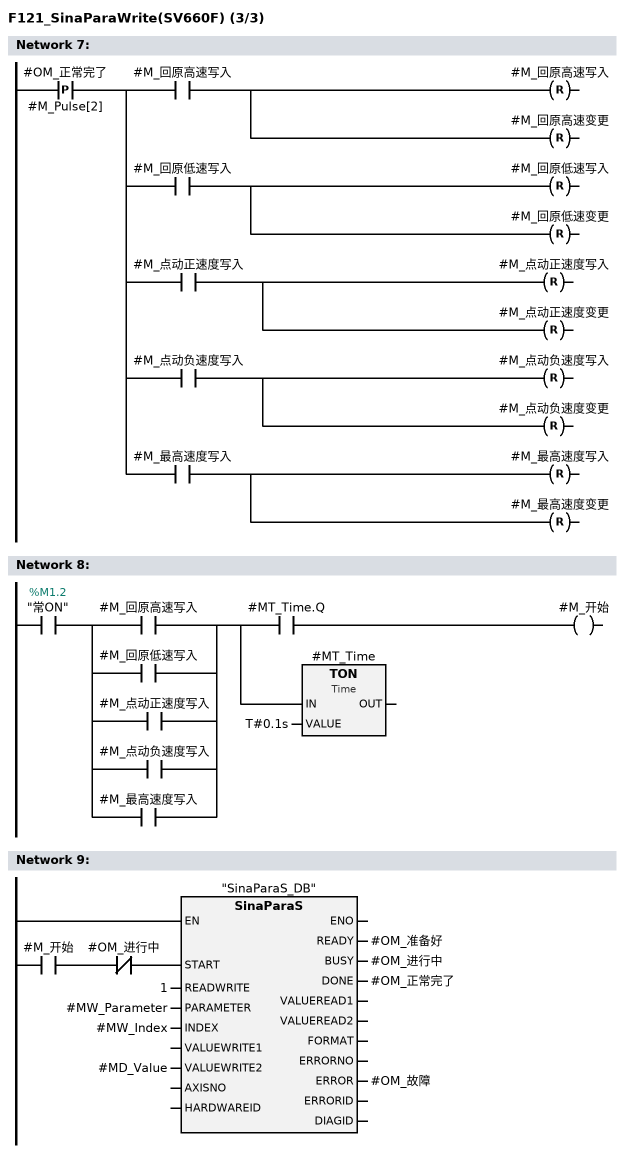
   RUNG wire#powerrail
      P_Contact(operand := #OM_正常完了, bit := #M_Pulse[2])
      wire#w1
      Contact( #M_回原高速写入 )
      wire#w2
      R_Coil( #M_回原高速写入 )
   END_RUNG
   RUNG wire#w2
      R_Coil( #M_回原高速变更 )
   END_RUNG
   RUNG wire#w1
      Contact( #M_回原低速写入 )
      wire#w3
      R_Coil( #M_回原低速写入 )
   END_RUNG
   RUNG wire#w3
      R_Coil( #M_回原低速变更 )
   END_RUNG
   RUNG wire#w1
      Contact( #M_点动正速度写入 )
      wire#w4
      R_Coil( #M_点动正速度写入 )
   END_RUNG
   RUNG wire#w4
      R_Coil( #M_点动正速度变更 )
   END_RUNG
   RUNG wire#w1
      Contact( #M_点动负速度写入 )
      wire#w5
      R_Coil( #M_点动负速度写入 )
   END_RUNG
   RUNG wire#w5
      R_Coil( #M_点动负速度变更 )
   END_RUNG
   RUNG wire#w1
      Contact( #M_最高速度写入 )
      wire#w6
      R_Coil( #M_最高速度写入 )
   END_RUNG
   RUNG wire#w6
      R_Coil( #M_最高速度变更 )
   END_RUNG
   // the same network as SCL:
   #_w1 := #OM_正常完了 AND NOT #M_Pulse[2];   // rising edge of #OM_正常完了
   #M_Pulse[2] := #OM_正常完了;
   #_w2 := #_w1 AND #M_回原高速写入;
   IF #_w2 THEN
       #M_回原高速写入 := FALSE;
       #M_回原高速变更 := FALSE;
   END_IF;
   #_w3 := #_w1 AND #M_回原低速写入;
   IF #_w3 THEN
       #M_回原低速写入 := FALSE;
       #M_回原低速变更 := FALSE;
   END_IF;
   #_w4 := #_w1 AND #M_点动正速度写入;
   IF #_w4 THEN
       #M_点动正速度写入 := FALSE;
       #M_点动正速度变更 := FALSE;
   END_IF;
   #_w5 := #_w1 AND #M_点动负速度写入;
   IF #_w5 THEN
       #M_点动负速度写入 := FALSE;
       #M_点动负速度变更 := FALSE;
   END_IF;
   #_w6 := #_w1 AND #M_最高速度写入;
   IF #_w6 THEN
       #M_最高速度写入 := FALSE;
       #M_最高速度变更 := FALSE;
   END_IF;
END_REGION

REGION Network 8
   #_w1 := "常ON" AND (#M_回原高速写入 OR #M_回原低速写入 OR #M_点动正速度写入 OR #M_点动负速度写入 OR #M_最高速度写入);
   #M_开始 := #_w1 AND #MT_Time.Q;
   #MT_Time.TON(IN := #_w1, PT := T#0.1s);   // TON coil
END_REGION

REGION Network 9
   RUNG wire#powerrail
      "SinaParaS_DB".SinaParaS(Start := wire#w1, ReadWrite := 1, Parameter := #MW_Parameter, Index := #MW_Index, ValueWrite1 :=, ValueWrite2 := #MD_Value, AxisNo :=, hardwareId :=, Ready => #OM_准备好, Busy => #OM_进行中, Done => #OM_正常完了, ValueRead1 =>, ValueRead2 =>, Format =>, ErrorNo =>, Error => #OM_故障, ErrorId =>, DiagId =>)
   END_RUNG
   RUNG wire#powerrail
      Contact( #M_开始 )
      I_Contact( #OM_进行中 )
   END_RUNG wire#w1
   // the same network as SCL:
   "SinaParaS_DB"(Start := #M_开始 AND NOT #OM_进行中,   // SinaParaS
                  ReadWrite := 1,
                  Parameter := #MW_Parameter,
                  Index := #MW_Index,
                  ValueWrite2 := #MD_Value,
                  Ready => #OM_准备好,
                  Busy => #OM_进行中,
                  Done => #OM_正常完了,
                  Error => #OM_故障);
END_REGION
END_FUNCTION_BLOCK

FUNCTION_BLOCK "F120_SinaPos(SV660F)"   // FB120, LAD
{ S7_Optimized_Access := 'TRUE' }
VERSION : 0.1
// 2024/2/4:第一版本V1.0，作者:wang
// stored: AutoNumber false, IsIECCheckEnabled false, IsRetainMemResEnabled false, MemoryReserve 100, SetENOAutomatically false, UDAEnableTagReadback false
   VAR_INPUT
      IW_手动模式 { ExternalAccessible := 'False'; ExternalVisible := 'False'; ExternalWritable := 'False'} : Bool;
      IW_运行条件 { ExternalAccessible := 'False'; ExternalVisible := 'False'; ExternalWritable := 'False'} : Array[1..8] of Bool;
      IM_使能 { ExternalAccessible := 'False'; ExternalVisible := 'False'; ExternalWritable := 'False'} : Bool;
      IM_回零 { ExternalAccessible := 'False'; ExternalVisible := 'False'; ExternalWritable := 'False'} : Bool;
      IM_绝对定位 { ExternalAccessible := 'False'; ExternalVisible := 'False'; ExternalWritable := 'False'} : Bool;
      IM_相对定位 { ExternalAccessible := 'False'; ExternalVisible := 'False'; ExternalWritable := 'False'} : Bool;
      "IM_JOG+" { ExternalAccessible := 'False'; ExternalVisible := 'False'; ExternalWritable := 'False'} : Bool;
      "IM_JOG-" { ExternalAccessible := 'False'; ExternalVisible := 'False'; ExternalWritable := 'False'} : Bool;
      IM_故障复位 { ExternalAccessible := 'False'; ExternalVisible := 'False'; ExternalWritable := 'False'} : Bool;
      ID_目标位置 { ExternalAccessible := 'False'; ExternalVisible := 'False'; ExternalWritable := 'False'} : DInt;
      ID_目标速度 { ExternalAccessible := 'False'; ExternalVisible := 'False'; ExternalWritable := 'False'} : DInt;
      "IW_速度加减倍率%" { ExternalAccessible := 'False'; ExternalVisible := 'False'; ExternalWritable := 'False'} : Array[1..3] of Int;
      ID_ConfigEpos { ExternalAccessible := 'False'; ExternalVisible := 'False'; ExternalWritable := 'False'} : DWord;
      ID_111报文标识符 { ExternalAccessible := 'False'; ExternalVisible := 'False'; ExternalWritable := 'False'} : HW_IO;
   END_VAR
   VAR_OUTPUT
      OM_准备好了 : Bool;
      OM_动作中 : Bool;
      OM_回零完了 : Bool;
      OM_轴报警 : Bool;
      OM_轴错误 : Bool;
      OD_当前位置 : DInt;
      OD_当前速度 : DInt;
      OW_运行模式 : Int;
      OW_EPSW1 : Word;
      OW_EPSW2 : Word;
      OW_轴报警码 : Word;
      OW_轴错误码 : Word;
      OW_库错误码 : Int;
      OW_调用错误码 : Word;
   END_VAR
   VAR
      MT_StartChk : IEC_TIMER;   // 启动延迟
   END_VAR
   VAR_TEMP
      M_停止 : Bool;
      M_暂停 : Bool;
      M_JOG指令 : Bool;
      M_回零指令 : Bool;
      M_绝对定位指令 : Bool;
      M_相对定位指令 : Bool;
      M_回零定位完Pls : Bool;
      M_绝对定位完Pls : Bool;
      M_相对定位完Pls : Bool;
      M_启动 : Bool;
      M_定位完了 : Bool;
      W_运行模式 : Int;
      M_Pulse : Array[1..20] of Bool;
      M_SerState : Bool;   // 伺服正常
      M_Busy : Bool;   // 伺服忙
      M_FLS_SW : Bool;   // 正极限
      M_RLS_SW : Bool;   // 负极限
   END_VAR
   // // IW_运行条件[1] : 共同条件
   // // IW_运行条件[2] : 回零条件
   // // IW_运行条件[3] : JOG正条件
   // // IW_运行条件[4] : JOG负条件
   // // IW_运行条件[5] : 定位正条件
   // // IW_运行条件[6] : 定位负条件
   // // IW_运行条件[7] : 预留
   // // IW_运行条件[8] : 预留
   VAR_TEMP   // added for the SCL form of the ladder/FBD networks
      _w1 : Bool;
      _w2 : Bool;
      _w3 : Bool;
      _w4 : Bool;
   END_VAR
BEGIN

REGION Network 1: 伺服状态条件
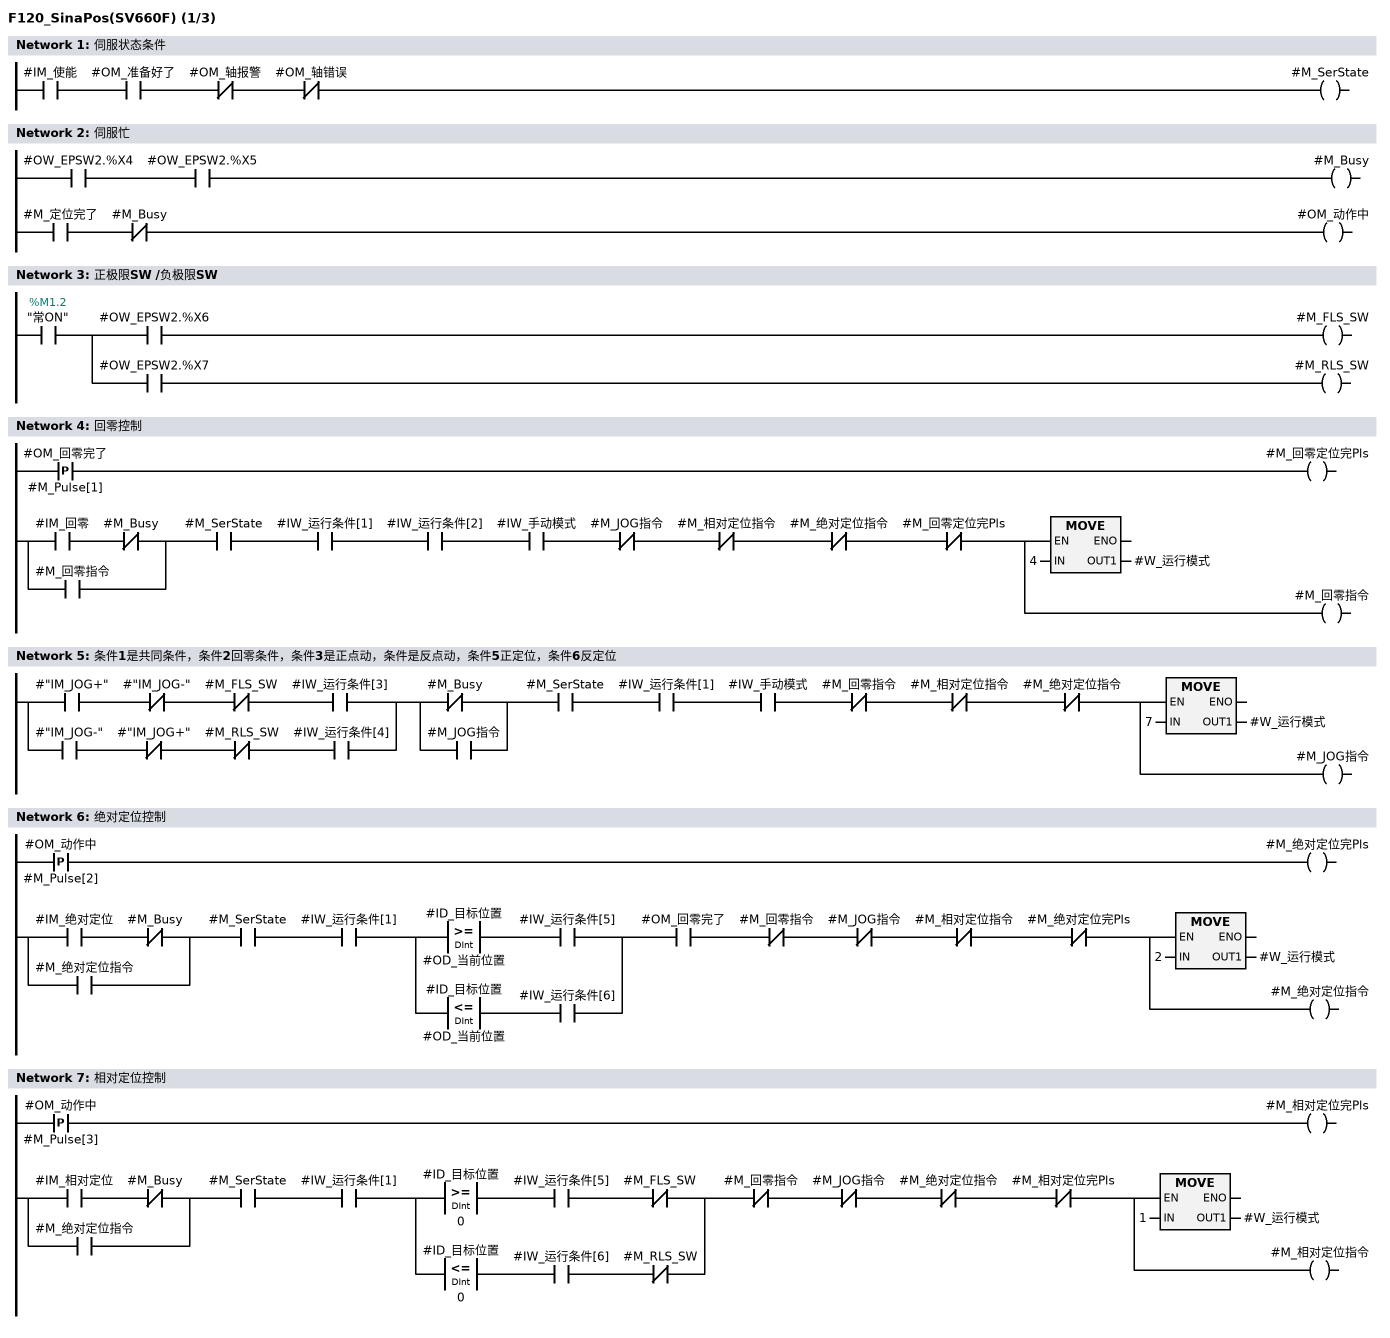
   RUNG wire#powerrail
      Contact( #IM_使能 )
      Contact( #OM_准备好了 )
      I_Contact( #OM_轴报警 )
      I_Contact( #OM_轴错误 )
      Coil( #M_SerState )
   END_RUNG
   // the same network as SCL:
   #M_SerState := #IM_使能 AND #OM_准备好了 AND NOT #OM_轴报警 AND NOT #OM_轴错误;
END_REGION

REGION Network 2: 伺服忙
   RUNG wire#powerrail
      Contact( #OW_EPSW2.%X4 )
      Contact( #OW_EPSW2.%X5 )
      Coil( #M_Busy )
   END_RUNG
   RUNG wire#powerrail
      Contact( #M_定位完了 )
      I_Contact( #M_Busy )
      Coil( #OM_动作中 )
   END_RUNG
   // the same network as SCL:
   #M_Busy := #OW_EPSW2.%X4 AND #OW_EPSW2.%X5;
   #OM_动作中 := #M_定位完了 AND NOT #M_Busy;
END_REGION

REGION Network 3: 正极限SW /负极限SW
   RUNG wire#powerrail
      Contact( "常ON" )
      wire#w1
      Contact( #OW_EPSW2.%X6 )
      Coil( #M_FLS_SW )
   END_RUNG
   RUNG wire#w1
      Contact( #OW_EPSW2.%X7 )
      Coil( #M_RLS_SW )
   END_RUNG
   // the same network as SCL:
   #M_FLS_SW := "常ON" AND #OW_EPSW2.%X6;
   #M_RLS_SW := "常ON" AND #OW_EPSW2.%X7;
END_REGION

REGION Network 4: 回零控制
   RUNG wire#powerrail
      P_Contact(operand := #OM_回零完了, bit := #M_Pulse[1])
      Coil( #M_回零定位完Pls )
   END_RUNG
   RUNG wire#powerrail
      Contact( #IM_回零 )
      I_Contact( #M_Busy )
      wire#w1
      Contact( #M_SerState )
      Contact( #IW_运行条件[1] )
      Contact( #IW_运行条件[2] )
      Contact( #IW_手动模式 )
      I_Contact( #M_JOG指令 )
      I_Contact( #M_相对定位指令 )
      I_Contact( #M_绝对定位指令 )
      I_Contact( #M_回零定位完Pls )
      wire#w2
      Move(in := 4, out1 => #W_运行模式)
   END_RUNG
   RUNG wire#powerrail
      Contact( #M_回零指令 )
   END_RUNG wire#w1
   RUNG wire#w2
      Coil( #M_回零指令 )
   END_RUNG
   // the same network as SCL:
   #_w1 := #OM_回零完了 AND NOT #M_Pulse[1];   // rising edge of #OM_回零完了
   #M_Pulse[1] := #OM_回零完了;
   #M_回零定位完Pls := #_w1;
   #_w2 := ((#IM_回零 AND NOT #M_Busy) OR #M_回零指令) AND #M_SerState AND #IW_运行条件[1] AND #IW_运行条件[2] AND #IW_手动模式 AND NOT #M_JOG指令 AND NOT #M_相对定位指令 AND NOT #M_绝对定位指令 AND NOT #M_回零定位完Pls;
   IF #_w2 THEN #W_运行模式 := 4; END_IF;
   #M_回零指令 := #_w2;
END_REGION

REGION Network 5: 条件1是共同条件，条件2回零条件，条件3是正点动，条件是反点动，条件5正定位，条件6反定位
   RUNG wire#powerrail
      Contact( #"IM_JOG+" )
      I_Contact( #"IM_JOG-" )
      I_Contact( #M_FLS_SW )
      Contact( #IW_运行条件[3] )
      wire#w1
      I_Contact( #M_Busy )
      wire#w2
      Contact( #M_SerState )
      Contact( #IW_运行条件[1] )
      Contact( #IW_手动模式 )
      I_Contact( #M_回零指令 )
      I_Contact( #M_相对定位指令 )
      I_Contact( #M_绝对定位指令 )
      wire#w3
      Move(in := 7, out1 => #W_运行模式)
   END_RUNG
   RUNG wire#powerrail
      Contact( #"IM_JOG-" )
      I_Contact( #"IM_JOG+" )
      I_Contact( #M_RLS_SW )
      Contact( #IW_运行条件[4] )
   END_RUNG wire#w1
   RUNG wire#w1
      Contact( #M_JOG指令 )
   END_RUNG wire#w2
   RUNG wire#w3
      Coil( #M_JOG指令 )
   END_RUNG
   // the same network as SCL:
   #_w1 := ((#"IM_JOG+" AND NOT #"IM_JOG-" AND NOT #M_FLS_SW AND #IW_运行条件[3]) OR (#"IM_JOG-" AND NOT #"IM_JOG+" AND NOT #M_RLS_SW AND #IW_运行条件[4])) AND (NOT #M_Busy OR #M_JOG指令) AND #M_SerState AND #IW_运行条件[1] AND #IW_手动模式 AND NOT #M_回零指令 AND NOT #M_相对定位指令 AND NOT #M_绝对定位指令;
   IF #_w1 THEN #W_运行模式 := 7; END_IF;
   #M_JOG指令 := #_w1;
END_REGION

REGION Network 6: 绝对定位控制
   RUNG wire#powerrail
      P_Contact(operand := #OM_动作中, bit := #M_Pulse[2])
      Coil( #M_绝对定位完Pls )
   END_RUNG
   RUNG wire#powerrail
      Contact( #IM_绝对定位 )
      I_Contact( #M_Busy )
      wire#w1
      Contact( #M_SerState )
      Contact( #IW_运行条件[1] )
      wire#w2
      { S7_Templates := "SrcType := DInt" } GE_Contact(in1 := #ID_目标位置, in2 := #OD_当前位置)
      Contact( #IW_运行条件[5] )
      wire#w3
      Contact( #OM_回零完了 )
      I_Contact( #M_回零指令 )
      I_Contact( #M_JOG指令 )
      I_Contact( #M_相对定位指令 )
      I_Contact( #M_绝对定位完Pls )
      wire#w4
      Move(in := 2, out1 => #W_运行模式)
   END_RUNG
   RUNG wire#powerrail
      Contact( #M_绝对定位指令 )
   END_RUNG wire#w1
   RUNG wire#w2
      { S7_Templates := "SrcType := DInt" } LE_Contact(in1 := #ID_目标位置, in2 := #OD_当前位置)
      Contact( #IW_运行条件[6] )
   END_RUNG wire#w3
   RUNG wire#w4
      Coil( #M_绝对定位指令 )
   END_RUNG
   // the same network as SCL:
   #_w1 := #OM_动作中 AND NOT #M_Pulse[2];   // rising edge of #OM_动作中
   #M_Pulse[2] := #OM_动作中;
   #M_绝对定位完Pls := #_w1;
   #_w2 := ((#IM_绝对定位 AND NOT #M_Busy) OR #M_绝对定位指令) AND #M_SerState AND #IW_运行条件[1] AND (((#ID_目标位置 >= #OD_当前位置) AND #IW_运行条件[5]) OR ((#ID_目标位置 <= #OD_当前位置) AND #IW_运行条件[6])) AND #OM_回零完了 AND NOT #M_回零指令 AND NOT #M_JOG指令 AND NOT #M_相对定位指令 AND NOT #M_绝对定位完Pls;
   IF #_w2 THEN #W_运行模式 := 2; END_IF;
   #M_绝对定位指令 := #_w2;
END_REGION

REGION Network 7: 相对定位控制
   RUNG wire#powerrail
      P_Contact(operand := #OM_动作中, bit := #M_Pulse[3])
      Coil( #M_相对定位完Pls )
   END_RUNG
   RUNG wire#powerrail
      Contact( #IM_相对定位 )
      I_Contact( #M_Busy )
      wire#w1
      Contact( #M_SerState )
      Contact( #IW_运行条件[1] )
      wire#w2
      { S7_Templates := "SrcType := DInt" } GE_Contact(in1 := #ID_目标位置, in2 := 0)
      Contact( #IW_运行条件[5] )
      I_Contact( #M_FLS_SW )
      wire#w3
      I_Contact( #M_回零指令 )
      I_Contact( #M_JOG指令 )
      I_Contact( #M_绝对定位指令 )
      I_Contact( #M_相对定位完Pls )
      wire#w4
      Move(in := 1, out1 => #W_运行模式)
   END_RUNG
   RUNG wire#powerrail
      Contact( #M_绝对定位指令 )
   END_RUNG wire#w1
   RUNG wire#w2
      { S7_Templates := "SrcType := DInt" } LE_Contact(in1 := #ID_目标位置, in2 := 0)
      Contact( #IW_运行条件[6] )
      I_Contact( #M_RLS_SW )
   END_RUNG wire#w3
   RUNG wire#w4
      Coil( #M_相对定位指令 )
   END_RUNG
   // the same network as SCL:
   #_w1 := #OM_动作中 AND NOT #M_Pulse[3];   // rising edge of #OM_动作中
   #M_Pulse[3] := #OM_动作中;
   #M_相对定位完Pls := #_w1;
   #_w2 := ((#IM_相对定位 AND NOT #M_Busy) OR #M_绝对定位指令) AND #M_SerState AND #IW_运行条件[1] AND (((#ID_目标位置 >= 0) AND #IW_运行条件[5] AND NOT #M_FLS_SW) OR ((#ID_目标位置 <= 0) AND #IW_运行条件[6] AND NOT #M_RLS_SW)) AND NOT #M_回零指令 AND NOT #M_JOG指令 AND NOT #M_绝对定位指令 AND NOT #M_相对定位完Pls;
   IF #_w2 THEN #W_运行模式 := 1; END_IF;
   #M_相对定位指令 := #_w2;
END_REGION

REGION Network 8: 控制启动
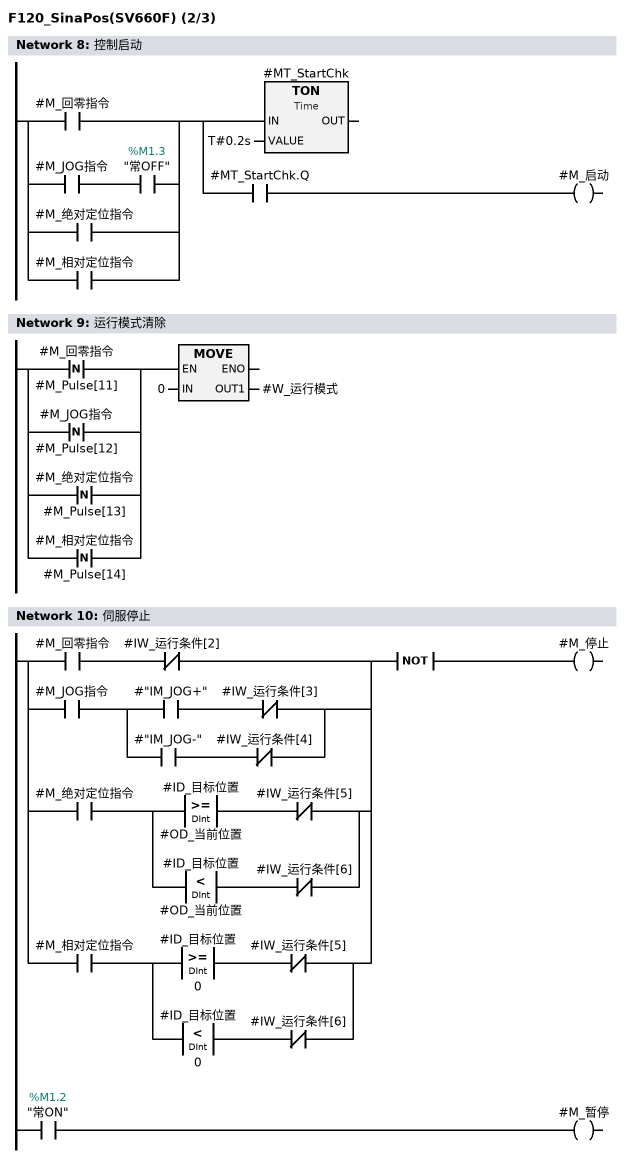
   #_w1 := #M_回零指令 OR (#M_JOG指令 AND "常OFF") OR #M_绝对定位指令 OR #M_相对定位指令;
   #MT_StartChk.TON(IN := #_w1, PT := T#0.2s);   // TON coil
   #M_启动 := #_w1 AND #MT_StartChk.Q;
END_REGION

REGION Network 9: 运行模式清除
   RUNG wire#powerrail
      N_Contact(operand := #M_回零指令, bit := #M_Pulse[11])
      wire#w1
      Move(in := 0, out1 => #W_运行模式)
   END_RUNG
   RUNG wire#powerrail
      N_Contact(operand := #M_JOG指令, bit := #M_Pulse[12])
   END_RUNG wire#w1
   RUNG wire#powerrail
      N_Contact(operand := #M_绝对定位指令, bit := #M_Pulse[13])
   END_RUNG wire#w1
   RUNG wire#powerrail
      N_Contact(operand := #M_相对定位指令, bit := #M_Pulse[14])
   END_RUNG wire#w1
   // the same network as SCL:
   #_w1 := NOT #M_回零指令 AND #M_Pulse[11];   // falling edge of #M_回零指令
   #M_Pulse[11] := #M_回零指令;
   #_w2 := NOT #M_JOG指令 AND #M_Pulse[12];   // falling edge of #M_JOG指令
   #M_Pulse[12] := #M_JOG指令;
   #_w3 := NOT #M_绝对定位指令 AND #M_Pulse[13];   // falling edge of #M_绝对定位指令
   #M_Pulse[13] := #M_绝对定位指令;
   #_w4 := NOT #M_相对定位指令 AND #M_Pulse[14];   // falling edge of #M_相对定位指令
   #M_Pulse[14] := #M_相对定位指令;
   IF #_w1 OR #_w2 OR #_w3 OR #_w4 THEN #W_运行模式 := 0; END_IF;
END_REGION

REGION Network 10: 伺服停止
   RUNG wire#powerrail
      Contact( #M_回零指令 )
      I_Contact( #IW_运行条件[2] )
      wire#w1
      Not()
      Coil( #M_停止 )
   END_RUNG
   RUNG wire#powerrail
      Contact( #M_JOG指令 )
      wire#w2
      Contact( #"IM_JOG+" )
      I_Contact( #IW_运行条件[3] )
   END_RUNG wire#w1
   RUNG wire#w2
      Contact( #"IM_JOG-" )
      I_Contact( #IW_运行条件[4] )
   END_RUNG wire#w1
   RUNG wire#powerrail
      Contact( #M_绝对定位指令 )
      wire#w3
      { S7_Templates := "SrcType := DInt" } GE_Contact(in1 := #ID_目标位置, in2 := #OD_当前位置)
      I_Contact( #IW_运行条件[5] )
   END_RUNG wire#w1
   RUNG wire#w3
      { S7_Templates := "SrcType := DInt" } LT_Contact(in1 := #ID_目标位置, in2 := #OD_当前位置)
      I_Contact( #IW_运行条件[6] )
   END_RUNG wire#w1
   RUNG wire#powerrail
      Contact( #M_相对定位指令 )
      wire#w4
      { S7_Templates := "SrcType := DInt" } GE_Contact(in1 := #ID_目标位置, in2 := 0)
      I_Contact( #IW_运行条件[5] )
   END_RUNG wire#w1
   RUNG wire#w4
      { S7_Templates := "SrcType := DInt" } LT_Contact(in1 := #ID_目标位置, in2 := 0)
      I_Contact( #IW_运行条件[6] )
   END_RUNG wire#w1
   RUNG wire#powerrail
      Contact( "常ON" )
      Coil( #M_暂停 )
   END_RUNG
   // the same network as SCL:
   #M_停止 := NOT ((#M_回零指令 AND NOT #IW_运行条件[2]) OR (#M_JOG指令 AND ((#"IM_JOG+" AND NOT #IW_运行条件[3]) OR (#"IM_JOG-" AND NOT #IW_运行条件[4]))) OR (#M_绝对定位指令 AND (((#ID_目标位置 >= #OD_当前位置) AND NOT #IW_运行条件[5]) OR ((#ID_目标位置 < #OD_当前位置) AND NOT #IW_运行条件[6]))) OR (#M_相对定位指令 AND (((#ID_目标位置 >= 0) AND NOT #IW_运行条件[5]) OR ((#ID_目标位置 < 0) AND NOT #IW_运行条件[6]))));
   #M_暂停 := "常ON";
END_REGION

REGION Network 11
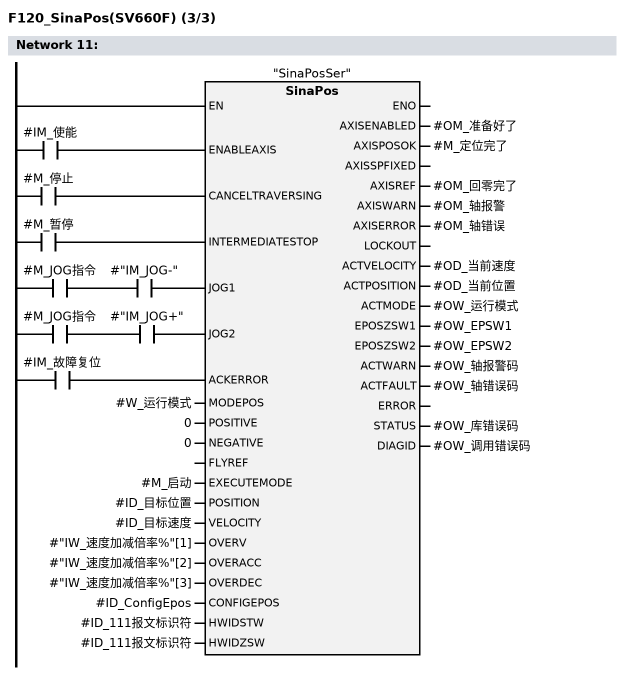
   RUNG wire#powerrail
      "SinaPosSer".SinaPos(EnableAxis := wire#w1, CancelTraversing := wire#w2, IntermediateStop := wire#w3, Jog1 := wire#w4, Jog2 := wire#w5, AckError := wire#w6, ModePos := #W_运行模式, Positive := 0, Negative := 0, FlyRef :=, ExecuteMode := #M_启动, Position := #ID_目标位置, Velocity := #ID_目标速度, OverV := #"IW_速度加减倍率%"[1], OverAcc := #"IW_速度加减倍率%"[2], OverDec := #"IW_速度加减倍率%"[3], ConfigEPos := #ID_ConfigEpos, HWIDSTW := #ID_111报文标识符, HWIDZSW := #ID_111报文标识符, AxisEnabled => #OM_准备好了, AxisPosOk => #M_定位完了, AxisSpFixed =>, AxisRef => #OM_回零完了, AxisWarn => #OM_轴报警, AxisError => #OM_轴错误, Lockout =>, ActVelocity => #OD_当前速度, ActPosition => #OD_当前位置, ActMode => #OW_运行模式, EPosZSW1 => #OW_EPSW1, EPosZSW2 => #OW_EPSW2, ActWarn => #OW_轴报警码, ActFault => #OW_轴错误码, Error =>, Status => #OW_库错误码, DiagId => #OW_调用错误码)
   END_RUNG
   RUNG wire#powerrail
      Contact( #IM_使能 )
   END_RUNG wire#w1
   RUNG wire#powerrail
      Contact( #M_停止 )
   END_RUNG wire#w2
   RUNG wire#powerrail
      Contact( #M_暂停 )
   END_RUNG wire#w3
   RUNG wire#powerrail
      Contact( #M_JOG指令 )
      Contact( #"IM_JOG-" )
   END_RUNG wire#w4
   RUNG wire#powerrail
      Contact( #M_JOG指令 )
      Contact( #"IM_JOG+" )
   END_RUNG wire#w5
   RUNG wire#powerrail
      Contact( #IM_故障复位 )
   END_RUNG wire#w6
   // the same network as SCL:
   "SinaPosSer"(EnableAxis := #IM_使能,   // SinaPos
                CancelTraversing := #M_停止,
                IntermediateStop := #M_暂停,
                Jog1 := #M_JOG指令 AND #"IM_JOG-",
                Jog2 := #M_JOG指令 AND #"IM_JOG+",
                AckError := #IM_故障复位,
                ModePos := #W_运行模式,
                Positive := 0,
                Negative := 0,
                ExecuteMode := #M_启动,
                Position := #ID_目标位置,
                Velocity := #ID_目标速度,
                OverV := #"IW_速度加减倍率%"[1],
                OverAcc := #"IW_速度加减倍率%"[2],
                OverDec := #"IW_速度加减倍率%"[3],
                ConfigEPos := #ID_ConfigEpos,
                HWIDSTW := #ID_111报文标识符,
                HWIDZSW := #ID_111报文标识符,
                AxisEnabled => #OM_准备好了,
                AxisPosOk => #M_定位完了,
                AxisRef => #OM_回零完了,
                AxisWarn => #OM_轴报警,
                AxisError => #OM_轴错误,
                ActVelocity => #OD_当前速度,
                ActPosition => #OD_当前位置,
                ActMode => #OW_运行模式,
                EPosZSW1 => #OW_EPSW1,
                EPosZSW2 => #OW_EPSW2,
                ActWarn => #OW_轴报警码,
                ActFault => #OW_轴错误码,
                Status => #OW_库错误码,
                DiagId => #OW_调用错误码);
END_REGION
END_FUNCTION_BLOCK

FUNCTION_BLOCK "K08_指示灯"   // FB8, LAD
{ S7_Optimized_Access := 'TRUE' }
VERSION : 0.1
// stored: AutoNumber false, IsIECCheckEnabled false, IsRetainMemResEnabled false, MemoryReserve 100, SetENOAutomatically false, UDAEnableTagReadback false
BEGIN

REGION Network 1: 自动灯
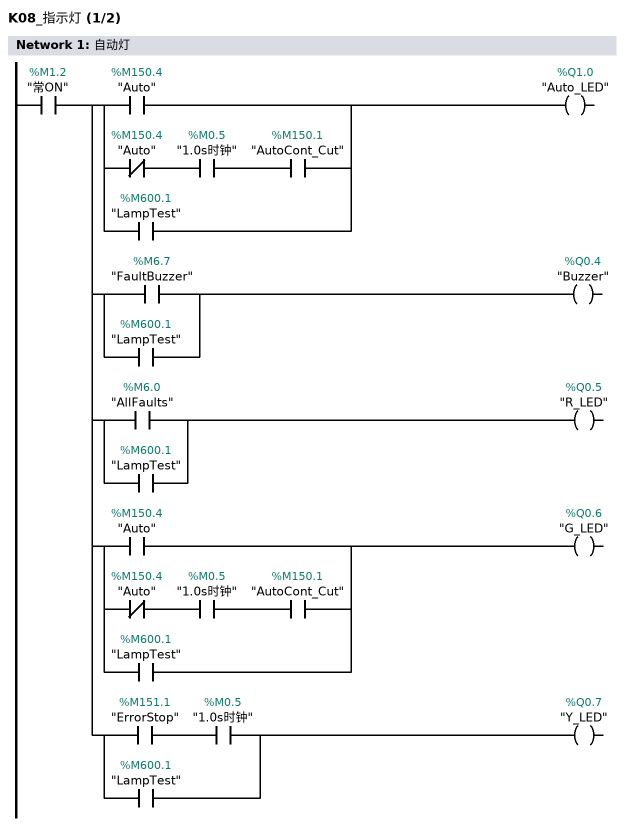
   RUNG wire#powerrail
      Contact( "常ON" )
      wire#w1
      Contact( "Auto" )
      wire#w2
      Coil( "Auto_LED" )
   END_RUNG
   RUNG wire#w1
      I_Contact( "Auto" )
      Contact( "1.0s时钟" )
      Contact( "AutoCont_Cut" )
   END_RUNG wire#w2
   RUNG wire#w1
      Contact( "LampTest" )
   END_RUNG wire#w2
   RUNG wire#w1
      Contact( "FaultBuzzer" )
      wire#w3
      Coil( "Buzzer" )
   END_RUNG
   RUNG wire#w1
      Contact( "LampTest" )
   END_RUNG wire#w3
   RUNG wire#w1
      Contact( "AllFaults" )
      wire#w4
      Coil( "R_LED" )
   END_RUNG
   RUNG wire#w1
      Contact( "LampTest" )
   END_RUNG wire#w4
   RUNG wire#w1
      Contact( "Auto" )
      wire#w5
      Coil( "G_LED" )
   END_RUNG
   RUNG wire#w1
      I_Contact( "Auto" )
      Contact( "1.0s时钟" )
      Contact( "AutoCont_Cut" )
   END_RUNG wire#w5
   RUNG wire#w1
      Contact( "LampTest" )
   END_RUNG wire#w5
   RUNG wire#w1
      Contact( "ErrorStop" )
      Contact( "1.0s时钟" )
      wire#w6
      Coil( "Y_LED" )
   END_RUNG
   RUNG wire#w1
      Contact( "LampTest" )
   END_RUNG wire#w6
   // the same network as SCL:
   "Auto_LED" := "常ON" AND ("Auto" OR (NOT "Auto" AND "1.0s时钟" AND "AutoCont_Cut") OR "LampTest");
   "Buzzer" := "常ON" AND ("FaultBuzzer" OR "LampTest");
   "R_LED" := "常ON" AND ("AllFaults" OR "LampTest");
   "G_LED" := "常ON" AND ("Auto" OR (NOT "Auto" AND "1.0s时钟" AND "AutoCont_Cut") OR "LampTest");
   "Y_LED" := "常ON" AND (("ErrorStop" AND "1.0s时钟") OR "LampTest");
END_REGION

REGION Network 2: 放行灯
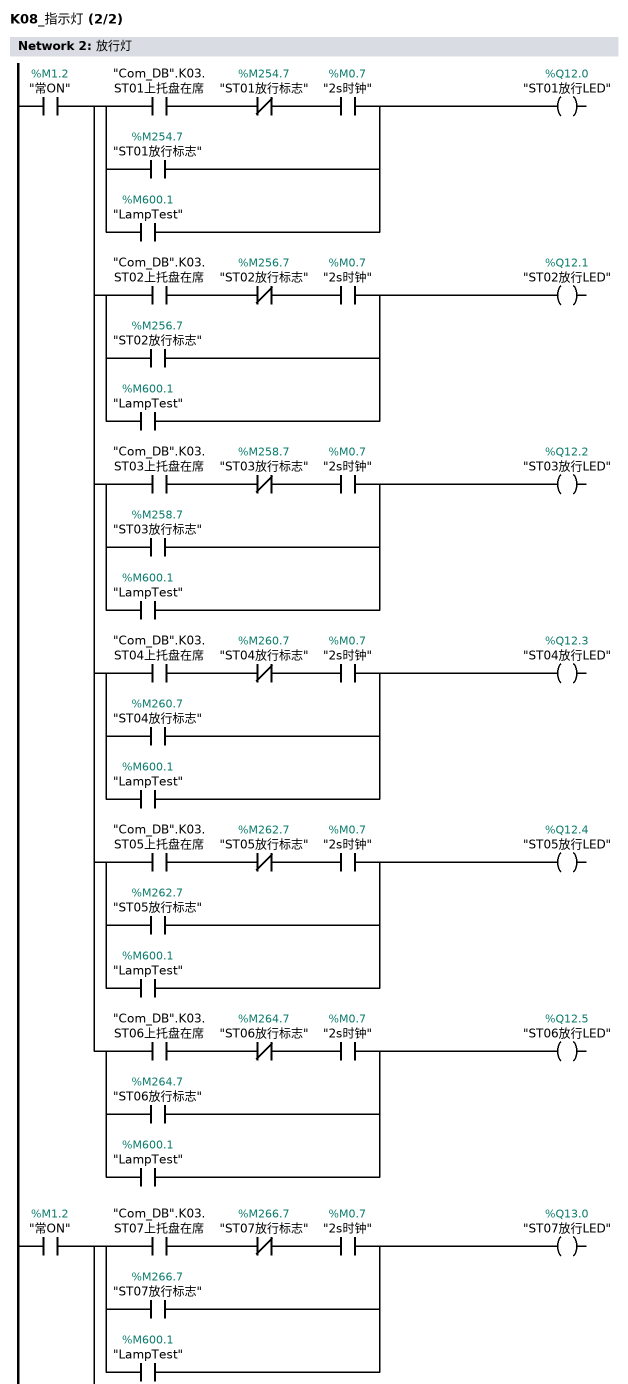
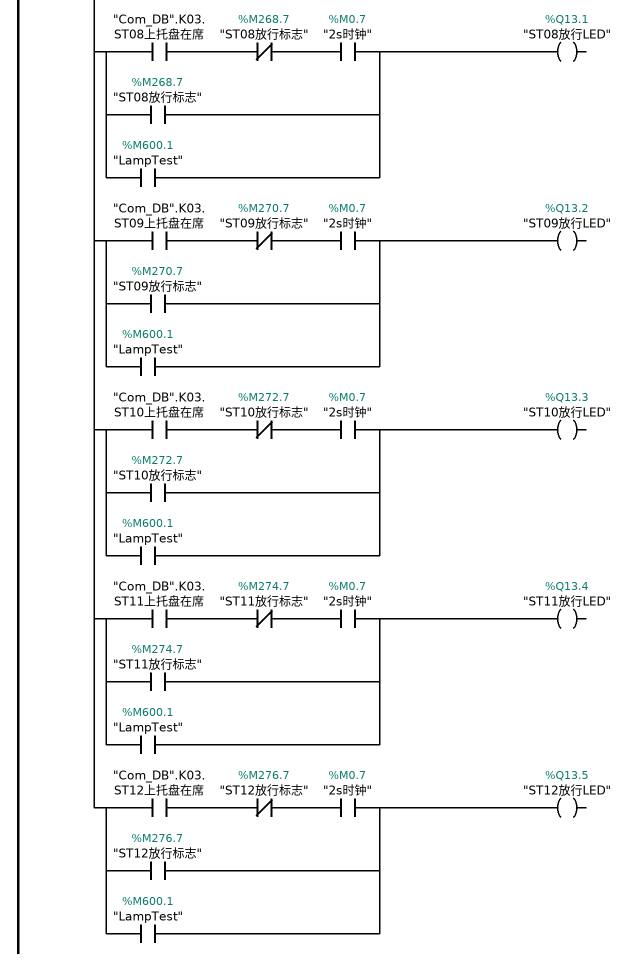
   RUNG wire#powerrail
      Contact( "常ON" )
      wire#w1
      Contact( "Com_DB".K03.ST01上托盘在席 )
      I_Contact( "ST01放行标志" )
      Contact( "2s时钟" )
      wire#w2
      Coil( "ST01放行LED" )
   END_RUNG
   RUNG wire#w1
      Contact( "ST01放行标志" )
   END_RUNG wire#w2
   RUNG wire#w1
      Contact( "LampTest" )
   END_RUNG wire#w2
   RUNG wire#w1
      Contact( "Com_DB".K03.ST02上托盘在席 )
      I_Contact( "ST02放行标志" )
      Contact( "2s时钟" )
      wire#w3
      Coil( "ST02放行LED" )
   END_RUNG
   RUNG wire#w1
      Contact( "ST02放行标志" )
   END_RUNG wire#w3
   RUNG wire#w1
      Contact( "LampTest" )
   END_RUNG wire#w3
   RUNG wire#w1
      Contact( "Com_DB".K03.ST03上托盘在席 )
      I_Contact( "ST03放行标志" )
      Contact( "2s时钟" )
      wire#w4
      Coil( "ST03放行LED" )
   END_RUNG
   RUNG wire#w1
      Contact( "ST03放行标志" )
   END_RUNG wire#w4
   RUNG wire#w1
      Contact( "LampTest" )
   END_RUNG wire#w4
   RUNG wire#w1
      Contact( "Com_DB".K03.ST04上托盘在席 )
      I_Contact( "ST04放行标志" )
      Contact( "2s时钟" )
      wire#w5
      Coil( "ST04放行LED" )
   END_RUNG
   RUNG wire#w1
      Contact( "ST04放行标志" )
   END_RUNG wire#w5
   RUNG wire#w1
      Contact( "LampTest" )
   END_RUNG wire#w5
   RUNG wire#w1
      Contact( "Com_DB".K03.ST05上托盘在席 )
      I_Contact( "ST05放行标志" )
      Contact( "2s时钟" )
      wire#w6
      Coil( "ST05放行LED" )
   END_RUNG
   RUNG wire#w1
      Contact( "ST05放行标志" )
   END_RUNG wire#w6
   RUNG wire#w1
      Contact( "LampTest" )
   END_RUNG wire#w6
   RUNG wire#w1
      Contact( "Com_DB".K03.ST06上托盘在席 )
      I_Contact( "ST06放行标志" )
      Contact( "2s时钟" )
      wire#w7
      Coil( "ST06放行LED" )
   END_RUNG
   RUNG wire#w1
      Contact( "ST06放行标志" )
   END_RUNG wire#w7
   RUNG wire#w1
      Contact( "LampTest" )
   END_RUNG wire#w7
   RUNG wire#powerrail
      Contact( "常ON" )
      wire#w8
      Contact( "Com_DB".K03.ST07上托盘在席 )
      I_Contact( "ST07放行标志" )
      Contact( "2s时钟" )
      wire#w9
      Coil( "ST07放行LED" )
   END_RUNG
   RUNG wire#w8
      Contact( "ST07放行标志" )
   END_RUNG wire#w9
   RUNG wire#w8
      Contact( "LampTest" )
   END_RUNG wire#w9
   RUNG wire#w8
      Contact( "Com_DB".K03.ST08上托盘在席 )
      I_Contact( "ST08放行标志" )
      Contact( "2s时钟" )
      wire#w10
      Coil( "ST08放行LED" )
   END_RUNG
   RUNG wire#w8
      Contact( "ST08放行标志" )
   END_RUNG wire#w10
   RUNG wire#w8
      Contact( "LampTest" )
   END_RUNG wire#w10
   RUNG wire#w8
      Contact( "Com_DB".K03.ST09上托盘在席 )
      I_Contact( "ST09放行标志" )
      Contact( "2s时钟" )
      wire#w11
      Coil( "ST09放行LED" )
   END_RUNG
   RUNG wire#w8
      Contact( "ST09放行标志" )
   END_RUNG wire#w11
   RUNG wire#w8
      Contact( "LampTest" )
   END_RUNG wire#w11
   RUNG wire#w8
      Contact( "Com_DB".K03.ST10上托盘在席 )
      I_Contact( "ST10放行标志" )
      Contact( "2s时钟" )
      wire#w12
      Coil( "ST10放行LED" )
   END_RUNG
   RUNG wire#w8
      Contact( "ST10放行标志" )
   END_RUNG wire#w12
   RUNG wire#w8
      Contact( "LampTest" )
   END_RUNG wire#w12
   RUNG wire#w8
      Contact( "Com_DB".K03.ST11上托盘在席 )
      I_Contact( "ST11放行标志" )
      Contact( "2s时钟" )
      wire#w13
      Coil( "ST11放行LED" )
   END_RUNG
   RUNG wire#w8
      Contact( "ST11放行标志" )
   END_RUNG wire#w13
   RUNG wire#w8
      Contact( "LampTest" )
   END_RUNG wire#w13
   RUNG wire#w8
      Contact( "Com_DB".K03.ST12上托盘在席 )
      I_Contact( "ST12放行标志" )
      Contact( "2s时钟" )
      wire#w14
      Coil( "ST12放行LED" )
   END_RUNG
   RUNG wire#w8
      Contact( "ST12放行标志" )
   END_RUNG wire#w14
   RUNG wire#w8
      Contact( "LampTest" )
   END_RUNG wire#w14
   // the same network as SCL:
   "ST01放行LED" := "常ON" AND (("Com_DB".K03.ST01上托盘在席 AND NOT "ST01放行标志" AND "2s时钟") OR "ST01放行标志" OR "LampTest");
   "ST02放行LED" := "常ON" AND (("Com_DB".K03.ST02上托盘在席 AND NOT "ST02放行标志" AND "2s时钟") OR "ST02放行标志" OR "LampTest");
   "ST03放行LED" := "常ON" AND (("Com_DB".K03.ST03上托盘在席 AND NOT "ST03放行标志" AND "2s时钟") OR "ST03放行标志" OR "LampTest");
   "ST04放行LED" := "常ON" AND (("Com_DB".K03.ST04上托盘在席 AND NOT "ST04放行标志" AND "2s时钟") OR "ST04放行标志" OR "LampTest");
   "ST05放行LED" := "常ON" AND (("Com_DB".K03.ST05上托盘在席 AND NOT "ST05放行标志" AND "2s时钟") OR "ST05放行标志" OR "LampTest");
   "ST06放行LED" := "常ON" AND (("Com_DB".K03.ST06上托盘在席 AND NOT "ST06放行标志" AND "2s时钟") OR "ST06放行标志" OR "LampTest");
   "ST07放行LED" := "常ON" AND (("Com_DB".K03.ST07上托盘在席 AND NOT "ST07放行标志" AND "2s时钟") OR "ST07放行标志" OR "LampTest");
   "ST08放行LED" := "常ON" AND (("Com_DB".K03.ST08上托盘在席 AND NOT "ST08放行标志" AND "2s时钟") OR "ST08放行标志" OR "LampTest");
   "ST09放行LED" := "常ON" AND (("Com_DB".K03.ST09上托盘在席 AND NOT "ST09放行标志" AND "2s时钟") OR "ST09放行标志" OR "LampTest");
   "ST10放行LED" := "常ON" AND (("Com_DB".K03.ST10上托盘在席 AND NOT "ST10放行标志" AND "2s时钟") OR "ST10放行标志" OR "LampTest");
   "ST11放行LED" := "常ON" AND (("Com_DB".K03.ST11上托盘在席 AND NOT "ST11放行标志" AND "2s时钟") OR "ST11放行标志" OR "LampTest");
   "ST12放行LED" := "常ON" AND (("Com_DB".K03.ST12上托盘在席 AND NOT "ST12放行标志" AND "2s时钟") OR "ST12放行标志" OR "LampTest");
END_REGION
END_FUNCTION_BLOCK

FUNCTION_BLOCK "K10_自动"   // FB10, LAD
{ S7_Optimized_Access := 'TRUE' }
VERSION : 0.1
// stored: AutoNumber false, IsIECCheckEnabled false, IsRetainMemResEnabled false, MemoryReserve 100, SetENOAutomatically false, UDAEnableTagReadback false
   VAR_TEMP
      M_OneStep : Bool;   // 单步运行
      M_Pluse : Array[1..10] of Bool;   // 脉冲
      "M_Init Pos1" : Bool;   // 初始位1
      "M_Init Pos2" : Bool;   // 初始位2
   END_VAR
   VAR_TEMP   // added for the SCL form of the ladder/FBD networks
      _w1 : Bool;
   END_VAR
BEGIN

REGION Network 1: 自动条件(立停)
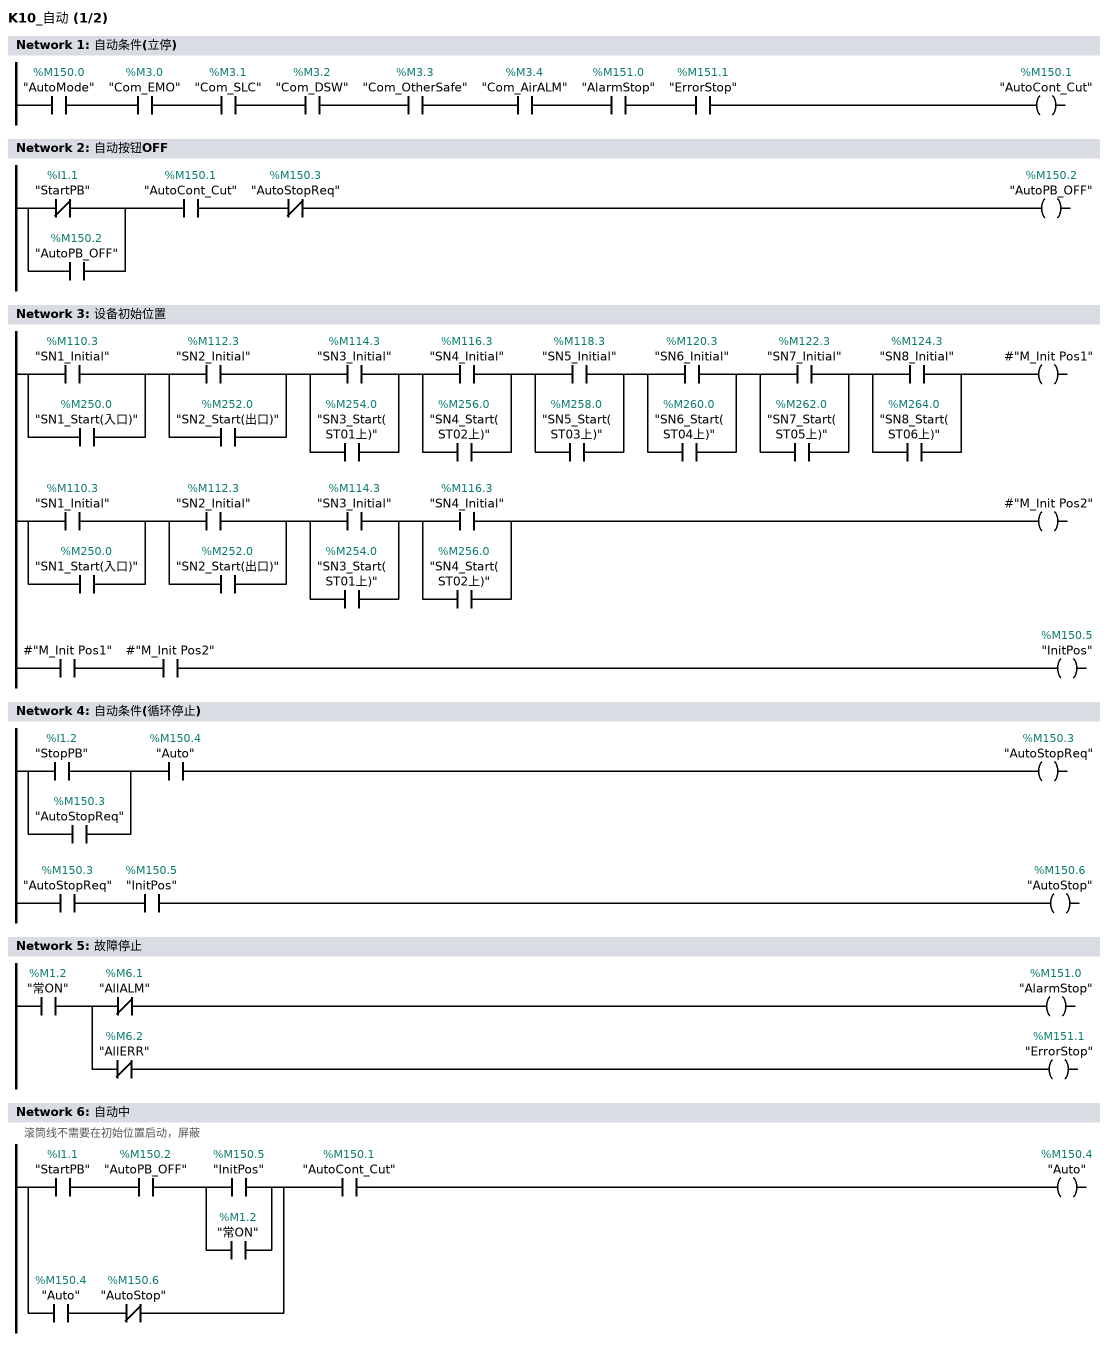
   RUNG wire#powerrail
      Contact( "AutoMode" )
      Contact( "Com_EMO" )
      Contact( "Com_SLC" )
      Contact( "Com_DSW" )
      Contact( "Com_OtherSafe" )
      Contact( "Com_AirALM" )
      Contact( "AlarmStop" )
      Contact( "ErrorStop" )
      Coil( "AutoCont_Cut" )
   END_RUNG
   // the same network as SCL:
   "AutoCont_Cut" := "AutoMode" AND "Com_EMO" AND "Com_SLC" AND "Com_DSW" AND "Com_OtherSafe" AND "Com_AirALM" AND "AlarmStop" AND "ErrorStop";
END_REGION

REGION Network 2: 自动按钮OFF
   RUNG wire#powerrail
      I_Contact( "StartPB" )
      wire#w1
      Contact( "AutoCont_Cut" )
      I_Contact( "AutoStopReq" )
      Coil( "AutoPB_OFF" )
   END_RUNG
   RUNG wire#powerrail
      Contact( "AutoPB_OFF" )
   END_RUNG wire#w1
   // the same network as SCL:
   "AutoPB_OFF" := (NOT "StartPB" OR "AutoPB_OFF") AND "AutoCont_Cut" AND NOT "AutoStopReq";
END_REGION

REGION Network 3: 设备初始位置
   RUNG wire#powerrail
      Contact( "SN1_Initial" )
      wire#w1
      Contact( "SN2_Initial" )
      wire#w2
      Contact( "SN3_Initial" )
      wire#w3
      Contact( "SN4_Initial" )
      wire#w4
      Contact( "SN5_Initial" )
      wire#w5
      Contact( "SN6_Initial" )
      wire#w6
      Contact( "SN7_Initial" )
      wire#w7
      Contact( "SN8_Initial" )
      wire#w8
      Coil( #"M_Init Pos1" )
   END_RUNG
   RUNG wire#powerrail
      Contact( "SN1_Start(入口)" )
   END_RUNG wire#w1
   RUNG wire#w1
      Contact( "SN2_Start(出口)" )
   END_RUNG wire#w2
   RUNG wire#w2
      Contact( "SN3_Start(ST01上)" )
   END_RUNG wire#w3
   RUNG wire#w3
      Contact( "SN4_Start(ST02上)" )
   END_RUNG wire#w4
   RUNG wire#w4
      Contact( "SN5_Start(ST03上)" )
   END_RUNG wire#w5
   RUNG wire#w5
      Contact( "SN6_Start(ST04上)" )
   END_RUNG wire#w6
   RUNG wire#w6
      Contact( "SN7_Start(ST05上)" )
   END_RUNG wire#w7
   RUNG wire#w7
      Contact( "SN8_Start(ST06上)" )
   END_RUNG wire#w8
   RUNG wire#powerrail
      Contact( "SN1_Initial" )
      wire#w9
      Contact( "SN2_Initial" )
      wire#w10
      Contact( "SN3_Initial" )
      wire#w11
      Contact( "SN4_Initial" )
      wire#w12
      Coil( #"M_Init Pos2" )
   END_RUNG
   RUNG wire#powerrail
      Contact( "SN1_Start(入口)" )
   END_RUNG wire#w9
   RUNG wire#w9
      Contact( "SN2_Start(出口)" )
   END_RUNG wire#w10
   RUNG wire#w10
      Contact( "SN3_Start(ST01上)" )
   END_RUNG wire#w11
   RUNG wire#w11
      Contact( "SN4_Start(ST02上)" )
   END_RUNG wire#w12
   RUNG wire#powerrail
      Contact( #"M_Init Pos1" )
      Contact( #"M_Init Pos2" )
      Coil( "InitPos" )
   END_RUNG
   // the same network as SCL:
   #"M_Init Pos1" := ("SN1_Initial" OR "SN1_Start(入口)") AND ("SN2_Initial" OR "SN2_Start(出口)") AND ("SN3_Initial" OR "SN3_Start(ST01上)") AND ("SN4_Initial" OR "SN4_Start(ST02上)") AND ("SN5_Initial" OR "SN5_Start(ST03上)") AND ("SN6_Initial" OR "SN6_Start(ST04上)") AND ("SN7_Initial" OR "SN7_Start(ST05上)") AND ("SN8_Initial" OR "SN8_Start(ST06上)");
   #"M_Init Pos2" := ("SN1_Initial" OR "SN1_Start(入口)") AND ("SN2_Initial" OR "SN2_Start(出口)") AND ("SN3_Initial" OR "SN3_Start(ST01上)") AND ("SN4_Initial" OR "SN4_Start(ST02上)");
   "InitPos" := #"M_Init Pos1" AND #"M_Init Pos2";
END_REGION

REGION Network 4: 自动条件(循环停止)
   RUNG wire#powerrail
      Contact( "StopPB" )
      wire#w1
      Contact( "Auto" )
      Coil( "AutoStopReq" )
   END_RUNG
   RUNG wire#powerrail
      Contact( "AutoStopReq" )
   END_RUNG wire#w1
   RUNG wire#powerrail
      Contact( "AutoStopReq" )
      Contact( "InitPos" )
      Coil( "AutoStop" )
   END_RUNG
   // the same network as SCL:
   "AutoStopReq" := ("StopPB" OR "AutoStopReq") AND "Auto";
   "AutoStop" := "AutoStopReq" AND "InitPos";
END_REGION

REGION Network 5: 故障停止
   RUNG wire#powerrail
      Contact( "常ON" )
      wire#w1
      I_Contact( "AllALM" )
      Coil( "AlarmStop" )
   END_RUNG
   RUNG wire#w1
      I_Contact( "AllERR" )
      Coil( "ErrorStop" )
   END_RUNG
   // the same network as SCL:
   "AlarmStop" := "常ON" AND NOT "AllALM";
   "ErrorStop" := "常ON" AND NOT "AllERR";
END_REGION

REGION Network 6: 自动中
   // 滚筒线不需要在初始位置启动，屏蔽
   RUNG wire#powerrail
      Contact( "StartPB" )
      Contact( "AutoPB_OFF" )
      wire#w1
      Contact( "InitPos" )
      wire#w2
      Contact( "AutoCont_Cut" )
      Coil( "Auto" )
   END_RUNG
   RUNG wire#w1
      Contact( "常ON" )
   END_RUNG wire#w2
   RUNG wire#powerrail
      Contact( "Auto" )
      I_Contact( "AutoStop" )
   END_RUNG wire#w2
   // the same network as SCL:
   "Auto" := (("StartPB" AND "AutoPB_OFF" AND ("InitPos" OR "常ON")) OR ("Auto" AND NOT "AutoStop")) AND "AutoCont_Cut";
END_REGION

REGION Network 7: 自动单步
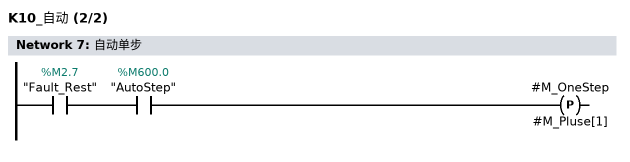
   #_w1 := "Fault_Rest" AND "AutoStep";
   #M_OneStep := #_w1 AND NOT #M_Pluse[1];   // rising edge
   #M_Pluse[1] := #_w1;
END_REGION
END_FUNCTION_BLOCK

FUNCTION_BLOCK "K11_入口自动"   // FB11, LAD
{ S7_Optimized_Access := 'TRUE' }
VERSION : 0.1
// stored: AutoNumber false, IsIECCheckEnabled false, IsRetainMemResEnabled false, MemoryReserve 100, SetENOAutomatically false, UDAEnableTagReadback false
   VAR_TEMP
      EN_提升机上升指令 : Array[1..8] of Bool;
      EN_提升机下降指令 : Array[1..8] of Bool;
      EN_阻挡上升指令 : Array[1..8] of Bool;
      EN_阻挡下降指令 : Array[1..8] of Bool;
   END_VAR
   VAR_TEMP   // added for the SCL form of the ladder/FBD networks
      _w1 : Bool;
   END_VAR
BEGIN

REGION Network 1: @SN1=入口部
END_REGION

REGION Network 2: @选择分支
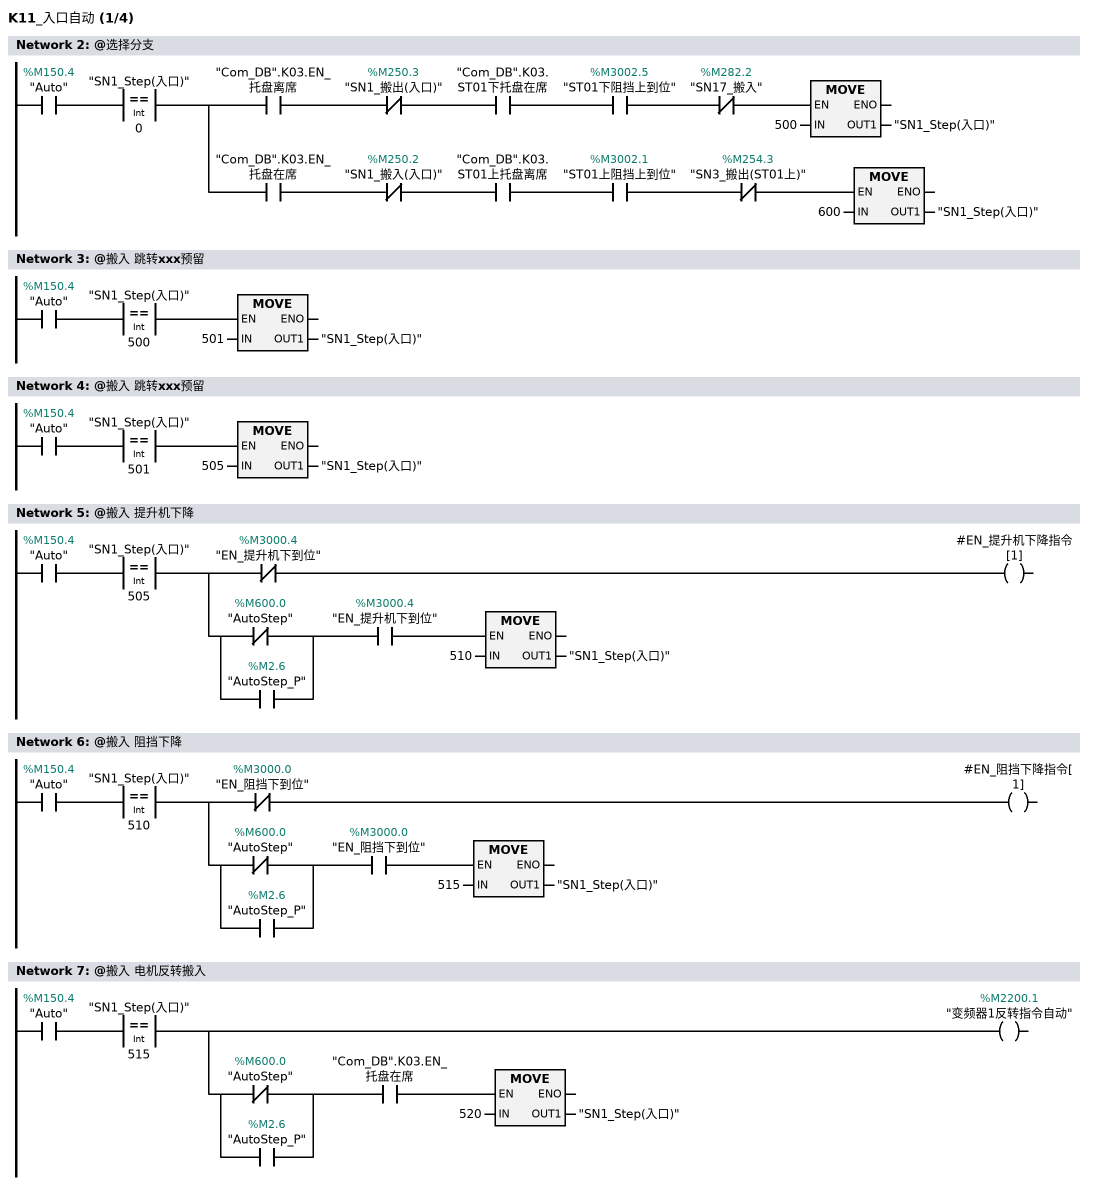
   RUNG wire#powerrail
      Contact( "Auto" )
      { S7_Templates := "SrcType := Int" } EQ_Contact(in1 := "SN1_Step(入口)", in2 := 0)
      wire#w1
      Contact( "Com_DB".K03.EN_托盘离席 )
      I_Contact( "SN1_搬出(入口)" )
      Contact( "Com_DB".K03.ST01下托盘在席 )
      Contact( "ST01下阻挡上到位" )
      I_Contact( "SN17_搬入" )
      Move(in := 500, out1 => "SN1_Step(入口)")
   END_RUNG
   RUNG wire#w1
      Contact( "Com_DB".K03.EN_托盘在席 )
      I_Contact( "SN1_搬入(入口)" )
      Contact( "Com_DB".K03.ST01上托盘离席 )
      Contact( "ST01上阻挡上到位" )
      I_Contact( "SN3_搬出(ST01上)" )
      Move(in := 600, out1 => "SN1_Step(入口)")
   END_RUNG
   // the same network as SCL:
   #_w1 := "Auto" AND ("SN1_Step(入口)" = 0);
   IF #_w1 AND "Com_DB".K03.EN_托盘离席 AND NOT "SN1_搬出(入口)" AND "Com_DB".K03.ST01下托盘在席 AND "ST01下阻挡上到位" AND NOT "SN17_搬入" THEN
       "SN1_Step(入口)" := 500;
   END_IF;
   IF #_w1 AND "Com_DB".K03.EN_托盘在席 AND NOT "SN1_搬入(入口)" AND "Com_DB".K03.ST01上托盘离席 AND "ST01上阻挡上到位" AND NOT "SN3_搬出(ST01上)" THEN
       "SN1_Step(入口)" := 600;
   END_IF;
END_REGION

REGION Network 3: @搬入 跳转xxx预留
   RUNG wire#powerrail
      Contact( "Auto" )
      { S7_Templates := "SrcType := Int" } EQ_Contact(in1 := "SN1_Step(入口)", in2 := 500)
      Move(in := 501, out1 => "SN1_Step(入口)")
   END_RUNG
   // the same network as SCL:
   IF "Auto" AND ("SN1_Step(入口)" = 500) THEN "SN1_Step(入口)" := 501; END_IF;
END_REGION

REGION Network 4: @搬入 跳转xxx预留
   RUNG wire#powerrail
      Contact( "Auto" )
      { S7_Templates := "SrcType := Int" } EQ_Contact(in1 := "SN1_Step(入口)", in2 := 501)
      Move(in := 505, out1 => "SN1_Step(入口)")
   END_RUNG
   // the same network as SCL:
   IF "Auto" AND ("SN1_Step(入口)" = 501) THEN "SN1_Step(入口)" := 505; END_IF;
END_REGION

REGION Network 5: @搬入 提升机下降
   RUNG wire#powerrail
      Contact( "Auto" )
      { S7_Templates := "SrcType := Int" } EQ_Contact(in1 := "SN1_Step(入口)", in2 := 505)
      wire#w1
      I_Contact( "EN_提升机下到位" )
      Coil( #EN_提升机下降指令[1] )
   END_RUNG
   RUNG wire#w1
      I_Contact( "AutoStep" )
      wire#w2
      Contact( "EN_提升机下到位" )
      Move(in := 510, out1 => "SN1_Step(入口)")
   END_RUNG
   RUNG wire#w1
      Contact( "AutoStep_P" )
   END_RUNG wire#w2
   // the same network as SCL:
   #_w1 := "Auto" AND ("SN1_Step(入口)" = 505);
   #EN_提升机下降指令[1] := #_w1 AND NOT "EN_提升机下到位";
   IF #_w1 AND (NOT "AutoStep" OR "AutoStep_P") AND "EN_提升机下到位" THEN "SN1_Step(入口)" := 510; END_IF;
END_REGION

REGION Network 6: @搬入 阻挡下降
   RUNG wire#powerrail
      Contact( "Auto" )
      { S7_Templates := "SrcType := Int" } EQ_Contact(in1 := "SN1_Step(入口)", in2 := 510)
      wire#w1
      I_Contact( "EN_阻挡下到位" )
      Coil( #EN_阻挡下降指令[1] )
   END_RUNG
   RUNG wire#w1
      I_Contact( "AutoStep" )
      wire#w2
      Contact( "EN_阻挡下到位" )
      Move(in := 515, out1 => "SN1_Step(入口)")
   END_RUNG
   RUNG wire#w1
      Contact( "AutoStep_P" )
   END_RUNG wire#w2
   // the same network as SCL:
   #_w1 := "Auto" AND ("SN1_Step(入口)" = 510);
   #EN_阻挡下降指令[1] := #_w1 AND NOT "EN_阻挡下到位";
   IF #_w1 AND (NOT "AutoStep" OR "AutoStep_P") AND "EN_阻挡下到位" THEN "SN1_Step(入口)" := 515; END_IF;
END_REGION

REGION Network 7: @搬入 电机反转搬入
   RUNG wire#powerrail
      Contact( "Auto" )
      { S7_Templates := "SrcType := Int" } EQ_Contact(in1 := "SN1_Step(入口)", in2 := 515)
      wire#w1
      Coil( "变频器1反转指令自动" )
   END_RUNG
   RUNG wire#w1
      I_Contact( "AutoStep" )
      wire#w2
      Contact( "Com_DB".K03.EN_托盘在席 )
      Move(in := 520, out1 => "SN1_Step(入口)")
   END_RUNG
   RUNG wire#w1
      Contact( "AutoStep_P" )
   END_RUNG wire#w2
   // the same network as SCL:
   "变频器1反转指令自动" := "Auto" AND ("SN1_Step(入口)" = 515);
   IF "变频器1反转指令自动" AND (NOT "AutoStep" OR "AutoStep_P") AND "Com_DB".K03.EN_托盘在席 THEN
       "SN1_Step(入口)" := 520;
   END_IF;
END_REGION

REGION Network 8: @搬入 阻挡上升
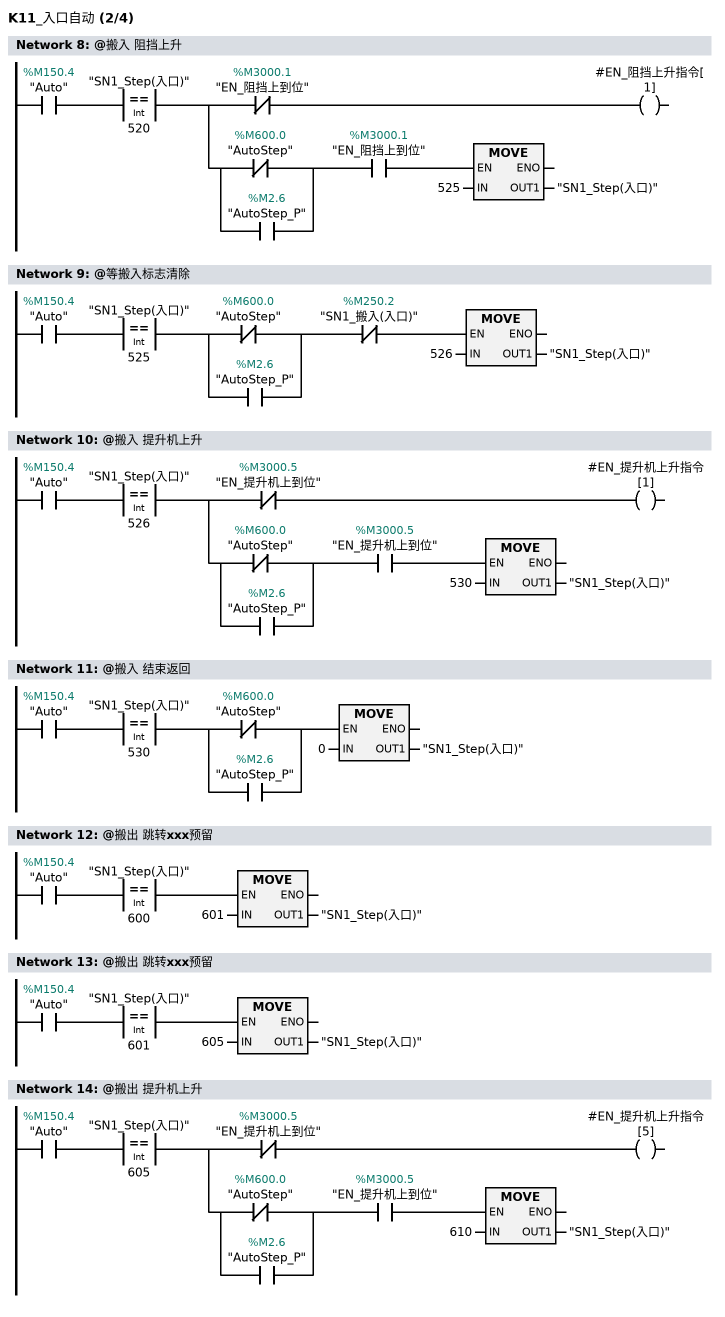
   RUNG wire#powerrail
      Contact( "Auto" )
      { S7_Templates := "SrcType := Int" } EQ_Contact(in1 := "SN1_Step(入口)", in2 := 520)
      wire#w1
      I_Contact( "EN_阻挡上到位" )
      Coil( #EN_阻挡上升指令[1] )
   END_RUNG
   RUNG wire#w1
      I_Contact( "AutoStep" )
      wire#w2
      Contact( "EN_阻挡上到位" )
      Move(in := 525, out1 => "SN1_Step(入口)")
   END_RUNG
   RUNG wire#w1
      Contact( "AutoStep_P" )
   END_RUNG wire#w2
   // the same network as SCL:
   #_w1 := "Auto" AND ("SN1_Step(入口)" = 520);
   #EN_阻挡上升指令[1] := #_w1 AND NOT "EN_阻挡上到位";
   IF #_w1 AND (NOT "AutoStep" OR "AutoStep_P") AND "EN_阻挡上到位" THEN "SN1_Step(入口)" := 525; END_IF;
END_REGION

REGION Network 9: @等搬入标志清除
   RUNG wire#powerrail
      Contact( "Auto" )
      { S7_Templates := "SrcType := Int" } EQ_Contact(in1 := "SN1_Step(入口)", in2 := 525)
      wire#w1
      I_Contact( "AutoStep" )
      wire#w2
      I_Contact( "SN1_搬入(入口)" )
      Move(in := 526, out1 => "SN1_Step(入口)")
   END_RUNG
   RUNG wire#w1
      Contact( "AutoStep_P" )
   END_RUNG wire#w2
   // the same network as SCL:
   IF "Auto" AND ("SN1_Step(入口)" = 525) AND (NOT "AutoStep" OR "AutoStep_P") AND NOT "SN1_搬入(入口)" THEN
       "SN1_Step(入口)" := 526;
   END_IF;
END_REGION

REGION Network 10: @搬入 提升机上升
   RUNG wire#powerrail
      Contact( "Auto" )
      { S7_Templates := "SrcType := Int" } EQ_Contact(in1 := "SN1_Step(入口)", in2 := 526)
      wire#w1
      I_Contact( "EN_提升机上到位" )
      Coil( #EN_提升机上升指令[1] )
   END_RUNG
   RUNG wire#w1
      I_Contact( "AutoStep" )
      wire#w2
      Contact( "EN_提升机上到位" )
      Move(in := 530, out1 => "SN1_Step(入口)")
   END_RUNG
   RUNG wire#w1
      Contact( "AutoStep_P" )
   END_RUNG wire#w2
   // the same network as SCL:
   #_w1 := "Auto" AND ("SN1_Step(入口)" = 526);
   #EN_提升机上升指令[1] := #_w1 AND NOT "EN_提升机上到位";
   IF #_w1 AND (NOT "AutoStep" OR "AutoStep_P") AND "EN_提升机上到位" THEN "SN1_Step(入口)" := 530; END_IF;
END_REGION

REGION Network 11: @搬入 结束返回
   RUNG wire#powerrail
      Contact( "Auto" )
      { S7_Templates := "SrcType := Int" } EQ_Contact(in1 := "SN1_Step(入口)", in2 := 530)
      wire#w1
      I_Contact( "AutoStep" )
      wire#w2
      Move(in := 0, out1 => "SN1_Step(入口)")
   END_RUNG
   RUNG wire#w1
      Contact( "AutoStep_P" )
   END_RUNG wire#w2
   // the same network as SCL:
   IF "Auto" AND ("SN1_Step(入口)" = 530) AND (NOT "AutoStep" OR "AutoStep_P") THEN
       "SN1_Step(入口)" := 0;
   END_IF;
END_REGION

REGION Network 12: @搬出 跳转xxx预留
   RUNG wire#powerrail
      Contact( "Auto" )
      { S7_Templates := "SrcType := Int" } EQ_Contact(in1 := "SN1_Step(入口)", in2 := 600)
      Move(in := 601, out1 => "SN1_Step(入口)")
   END_RUNG
   // the same network as SCL:
   IF "Auto" AND ("SN1_Step(入口)" = 600) THEN "SN1_Step(入口)" := 601; END_IF;
END_REGION

REGION Network 13: @搬出 跳转xxx预留
   RUNG wire#powerrail
      Contact( "Auto" )
      { S7_Templates := "SrcType := Int" } EQ_Contact(in1 := "SN1_Step(入口)", in2 := 601)
      Move(in := 605, out1 => "SN1_Step(入口)")
   END_RUNG
   // the same network as SCL:
   IF "Auto" AND ("SN1_Step(入口)" = 601) THEN "SN1_Step(入口)" := 605; END_IF;
END_REGION

REGION Network 14: @搬出 提升机上升
   RUNG wire#powerrail
      Contact( "Auto" )
      { S7_Templates := "SrcType := Int" } EQ_Contact(in1 := "SN1_Step(入口)", in2 := 605)
      wire#w1
      I_Contact( "EN_提升机上到位" )
      Coil( #EN_提升机上升指令[5] )
   END_RUNG
   RUNG wire#w1
      I_Contact( "AutoStep" )
      wire#w2
      Contact( "EN_提升机上到位" )
      Move(in := 610, out1 => "SN1_Step(入口)")
   END_RUNG
   RUNG wire#w1
      Contact( "AutoStep_P" )
   END_RUNG wire#w2
   // the same network as SCL:
   #_w1 := "Auto" AND ("SN1_Step(入口)" = 605);
   #EN_提升机上升指令[5] := #_w1 AND NOT "EN_提升机上到位";
   IF #_w1 AND (NOT "AutoStep" OR "AutoStep_P") AND "EN_提升机上到位" THEN "SN1_Step(入口)" := 610; END_IF;
END_REGION

REGION Network 15: @搬出 阻挡下降
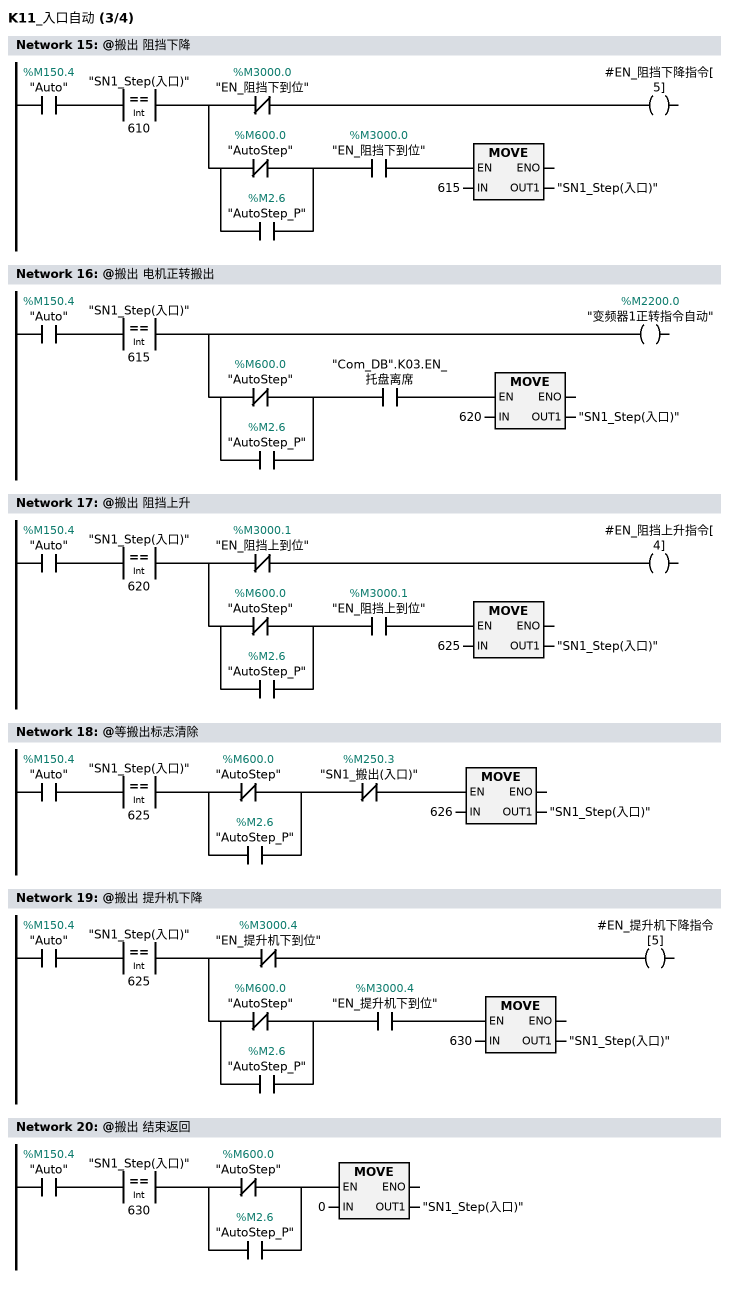
   RUNG wire#powerrail
      Contact( "Auto" )
      { S7_Templates := "SrcType := Int" } EQ_Contact(in1 := "SN1_Step(入口)", in2 := 610)
      wire#w1
      I_Contact( "EN_阻挡下到位" )
      Coil( #EN_阻挡下降指令[5] )
   END_RUNG
   RUNG wire#w1
      I_Contact( "AutoStep" )
      wire#w2
      Contact( "EN_阻挡下到位" )
      Move(in := 615, out1 => "SN1_Step(入口)")
   END_RUNG
   RUNG wire#w1
      Contact( "AutoStep_P" )
   END_RUNG wire#w2
   // the same network as SCL:
   #_w1 := "Auto" AND ("SN1_Step(入口)" = 610);
   #EN_阻挡下降指令[5] := #_w1 AND NOT "EN_阻挡下到位";
   IF #_w1 AND (NOT "AutoStep" OR "AutoStep_P") AND "EN_阻挡下到位" THEN "SN1_Step(入口)" := 615; END_IF;
END_REGION

REGION Network 16: @搬出 电机正转搬出
   RUNG wire#powerrail
      Contact( "Auto" )
      { S7_Templates := "SrcType := Int" } EQ_Contact(in1 := "SN1_Step(入口)", in2 := 615)
      wire#w1
      Coil( "变频器1正转指令自动" )
   END_RUNG
   RUNG wire#w1
      I_Contact( "AutoStep" )
      wire#w2
      Contact( "Com_DB".K03.EN_托盘离席 )
      Move(in := 620, out1 => "SN1_Step(入口)")
   END_RUNG
   RUNG wire#w1
      Contact( "AutoStep_P" )
   END_RUNG wire#w2
   // the same network as SCL:
   "变频器1正转指令自动" := "Auto" AND ("SN1_Step(入口)" = 615);
   IF "变频器1正转指令自动" AND (NOT "AutoStep" OR "AutoStep_P") AND "Com_DB".K03.EN_托盘离席 THEN
       "SN1_Step(入口)" := 620;
   END_IF;
END_REGION

REGION Network 17: @搬出 阻挡上升
   RUNG wire#powerrail
      Contact( "Auto" )
      { S7_Templates := "SrcType := Int" } EQ_Contact(in1 := "SN1_Step(入口)", in2 := 620)
      wire#w1
      I_Contact( "EN_阻挡上到位" )
      Coil( #EN_阻挡上升指令[4] )
   END_RUNG
   RUNG wire#w1
      I_Contact( "AutoStep" )
      wire#w2
      Contact( "EN_阻挡上到位" )
      Move(in := 625, out1 => "SN1_Step(入口)")
   END_RUNG
   RUNG wire#w1
      Contact( "AutoStep_P" )
   END_RUNG wire#w2
   // the same network as SCL:
   #_w1 := "Auto" AND ("SN1_Step(入口)" = 620);
   #EN_阻挡上升指令[4] := #_w1 AND NOT "EN_阻挡上到位";
   IF #_w1 AND (NOT "AutoStep" OR "AutoStep_P") AND "EN_阻挡上到位" THEN "SN1_Step(入口)" := 625; END_IF;
END_REGION

REGION Network 18: @等搬出标志清除
   RUNG wire#powerrail
      Contact( "Auto" )
      { S7_Templates := "SrcType := Int" } EQ_Contact(in1 := "SN1_Step(入口)", in2 := 625)
      wire#w1
      I_Contact( "AutoStep" )
      wire#w2
      I_Contact( "SN1_搬出(入口)" )
      Move(in := 626, out1 => "SN1_Step(入口)")
   END_RUNG
   RUNG wire#w1
      Contact( "AutoStep_P" )
   END_RUNG wire#w2
   // the same network as SCL:
   IF "Auto" AND ("SN1_Step(入口)" = 625) AND (NOT "AutoStep" OR "AutoStep_P") AND NOT "SN1_搬出(入口)" THEN
       "SN1_Step(入口)" := 626;
   END_IF;
END_REGION

REGION Network 19: @搬出 提升机下降
   RUNG wire#powerrail
      Contact( "Auto" )
      { S7_Templates := "SrcType := Int" } EQ_Contact(in1 := "SN1_Step(入口)", in2 := 625)
      wire#w1
      I_Contact( "EN_提升机下到位" )
      Coil( #EN_提升机下降指令[5] )
   END_RUNG
   RUNG wire#w1
      I_Contact( "AutoStep" )
      wire#w2
      Contact( "EN_提升机下到位" )
      Move(in := 630, out1 => "SN1_Step(入口)")
   END_RUNG
   RUNG wire#w1
      Contact( "AutoStep_P" )
   END_RUNG wire#w2
   // the same network as SCL:
   #_w1 := "Auto" AND ("SN1_Step(入口)" = 625);
   #EN_提升机下降指令[5] := #_w1 AND NOT "EN_提升机下到位";
   IF #_w1 AND (NOT "AutoStep" OR "AutoStep_P") AND "EN_提升机下到位" THEN "SN1_Step(入口)" := 630; END_IF;
END_REGION

REGION Network 20: @搬出 结束返回
   RUNG wire#powerrail
      Contact( "Auto" )
      { S7_Templates := "SrcType := Int" } EQ_Contact(in1 := "SN1_Step(入口)", in2 := 630)
      wire#w1
      I_Contact( "AutoStep" )
      wire#w2
      Move(in := 0, out1 => "SN1_Step(入口)")
   END_RUNG
   RUNG wire#w1
      Contact( "AutoStep_P" )
   END_RUNG wire#w2
   // the same network as SCL:
   IF "Auto" AND ("SN1_Step(入口)" = 630) AND (NOT "AutoStep" OR "AutoStep_P") THEN
       "SN1_Step(入口)" := 0;
   END_IF;
END_REGION

REGION Network 21: 控制输出
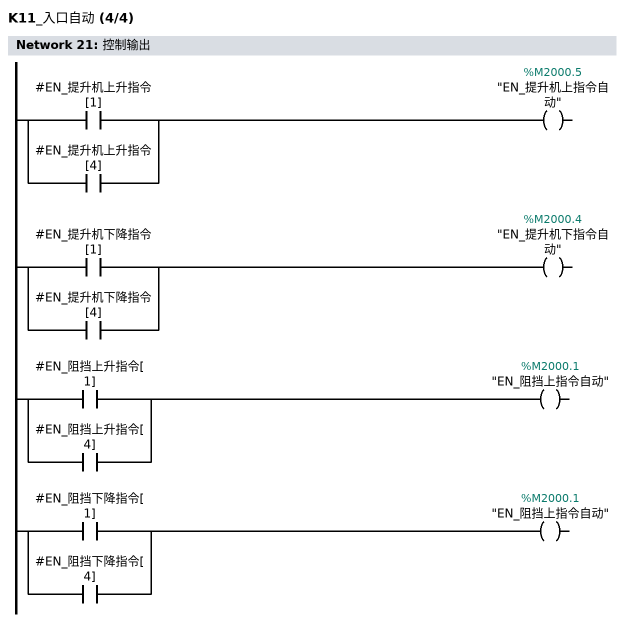
   RUNG wire#powerrail
      Contact( #EN_提升机上升指令[1] )
      wire#w1
      Coil( "EN_提升机上指令自动" )
   END_RUNG
   RUNG wire#powerrail
      Contact( #EN_提升机上升指令[4] )
   END_RUNG wire#w1
   RUNG wire#powerrail
      Contact( #EN_提升机下降指令[1] )
      wire#w2
      Coil( "EN_提升机下指令自动" )
   END_RUNG
   RUNG wire#powerrail
      Contact( #EN_提升机下降指令[4] )
   END_RUNG wire#w2
   RUNG wire#powerrail
      Contact( #EN_阻挡上升指令[1] )
      wire#w3
      Coil( "EN_阻挡上指令自动" )
   END_RUNG
   RUNG wire#powerrail
      Contact( #EN_阻挡上升指令[4] )
   END_RUNG wire#w3
   RUNG wire#powerrail
      Contact( #EN_阻挡下降指令[1] )
      wire#w4
      Coil( "EN_阻挡上指令自动" )
   END_RUNG
   RUNG wire#powerrail
      Contact( #EN_阻挡下降指令[4] )
   END_RUNG wire#w4
   // the same network as SCL:
   "EN_提升机上指令自动" := #EN_提升机上升指令[1] OR #EN_提升机上升指令[4];
   "EN_提升机下指令自动" := #EN_提升机下降指令[1] OR #EN_提升机下降指令[4];
   "EN_阻挡上指令自动" := #EN_阻挡上升指令[1] OR #EN_阻挡上升指令[4];
   "EN_阻挡上指令自动" := #EN_阻挡下降指令[1] OR #EN_阻挡下降指令[4];
END_REGION
END_FUNCTION_BLOCK

FUNCTION_BLOCK "K12_出口自动"   // FB12, LAD
{ S7_Optimized_Access := 'TRUE' }
VERSION : 0.1
// stored: AutoNumber false, IsIECCheckEnabled false, IsRetainMemResEnabled false, MemoryReserve 100, SetENOAutomatically false, UDAEnableTagReadback false
   VAR_TEMP
      EX_提升机上升指令 : Array[1..8] of Bool;
      EX_提升机下降指令 : Array[1..8] of Bool;
      EX_阻挡上升指令 : Array[1..8] of Bool;
      EX_阻挡下降指令 : Array[1..8] of Bool;
   END_VAR
   VAR_TEMP   // added for the SCL form of the ladder/FBD networks
      _w1 : Bool;
   END_VAR
BEGIN

REGION Network 1: @SN2=出口部
END_REGION

REGION Network 2: @选择分支
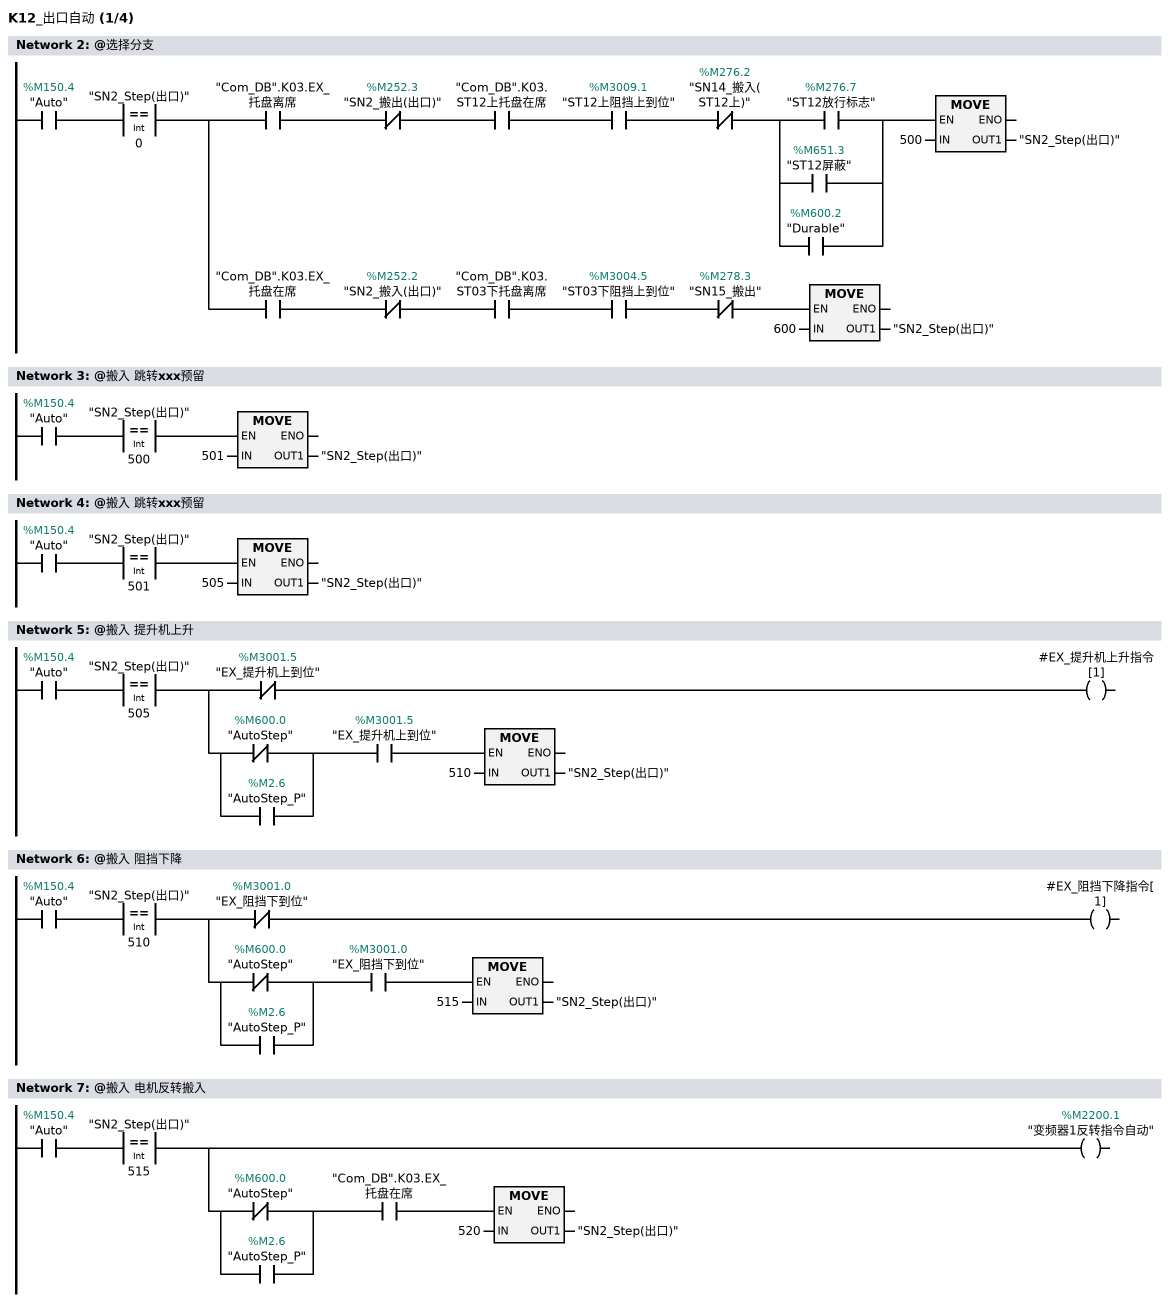
   RUNG wire#powerrail
      Contact( "Auto" )
      { S7_Templates := "SrcType := Int" } EQ_Contact(in1 := "SN2_Step(出口)", in2 := 0)
      wire#w1
      Contact( "Com_DB".K03.EX_托盘离席 )
      I_Contact( "SN2_搬出(出口)" )
      Contact( "Com_DB".K03.ST12上托盘在席 )
      Contact( "ST12上阻挡上到位" )
      I_Contact( "SN14_搬入(ST12上)" )
      wire#w2
      Contact( "ST12放行标志" )
      wire#w3
      Move(in := 500, out1 => "SN2_Step(出口)")
   END_RUNG
   RUNG wire#w2
      Contact( "ST12屏蔽" )
   END_RUNG wire#w3
   RUNG wire#w2
      Contact( "Durable" )
   END_RUNG wire#w3
   RUNG wire#w1
      Contact( "Com_DB".K03.EX_托盘在席 )
      I_Contact( "SN2_搬入(出口)" )
      Contact( "Com_DB".K03.ST03下托盘离席 )
      Contact( "ST03下阻挡上到位" )
      I_Contact( "SN15_搬出" )
      Move(in := 600, out1 => "SN2_Step(出口)")
   END_RUNG
   // the same network as SCL:
   #_w1 := "Auto" AND ("SN2_Step(出口)" = 0);
   IF #_w1 AND "Com_DB".K03.EX_托盘离席 AND NOT "SN2_搬出(出口)" AND "Com_DB".K03.ST12上托盘在席 AND "ST12上阻挡上到位" AND NOT "SN14_搬入(ST12上)" AND ("ST12放行标志" OR "ST12屏蔽" OR "Durable") THEN
       "SN2_Step(出口)" := 500;
   END_IF;
   IF #_w1 AND "Com_DB".K03.EX_托盘在席 AND NOT "SN2_搬入(出口)" AND "Com_DB".K03.ST03下托盘离席 AND "ST03下阻挡上到位" AND NOT "SN15_搬出" THEN
       "SN2_Step(出口)" := 600;
   END_IF;
END_REGION

REGION Network 3: @搬入 跳转xxx预留
   RUNG wire#powerrail
      Contact( "Auto" )
      { S7_Templates := "SrcType := Int" } EQ_Contact(in1 := "SN2_Step(出口)", in2 := 500)
      Move(in := 501, out1 => "SN2_Step(出口)")
   END_RUNG
   // the same network as SCL:
   IF "Auto" AND ("SN2_Step(出口)" = 500) THEN "SN2_Step(出口)" := 501; END_IF;
END_REGION

REGION Network 4: @搬入 跳转xxx预留
   RUNG wire#powerrail
      Contact( "Auto" )
      { S7_Templates := "SrcType := Int" } EQ_Contact(in1 := "SN2_Step(出口)", in2 := 501)
      Move(in := 505, out1 => "SN2_Step(出口)")
   END_RUNG
   // the same network as SCL:
   IF "Auto" AND ("SN2_Step(出口)" = 501) THEN "SN2_Step(出口)" := 505; END_IF;
END_REGION

REGION Network 5: @搬入 提升机上升
   RUNG wire#powerrail
      Contact( "Auto" )
      { S7_Templates := "SrcType := Int" } EQ_Contact(in1 := "SN2_Step(出口)", in2 := 505)
      wire#w1
      I_Contact( "EX_提升机上到位" )
      Coil( #EX_提升机上升指令[1] )
   END_RUNG
   RUNG wire#w1
      I_Contact( "AutoStep" )
      wire#w2
      Contact( "EX_提升机上到位" )
      Move(in := 510, out1 => "SN2_Step(出口)")
   END_RUNG
   RUNG wire#w1
      Contact( "AutoStep_P" )
   END_RUNG wire#w2
   // the same network as SCL:
   #_w1 := "Auto" AND ("SN2_Step(出口)" = 505);
   #EX_提升机上升指令[1] := #_w1 AND NOT "EX_提升机上到位";
   IF #_w1 AND (NOT "AutoStep" OR "AutoStep_P") AND "EX_提升机上到位" THEN "SN2_Step(出口)" := 510; END_IF;
END_REGION

REGION Network 6: @搬入 阻挡下降
   RUNG wire#powerrail
      Contact( "Auto" )
      { S7_Templates := "SrcType := Int" } EQ_Contact(in1 := "SN2_Step(出口)", in2 := 510)
      wire#w1
      I_Contact( "EX_阻挡下到位" )
      Coil( #EX_阻挡下降指令[1] )
   END_RUNG
   RUNG wire#w1
      I_Contact( "AutoStep" )
      wire#w2
      Contact( "EX_阻挡下到位" )
      Move(in := 515, out1 => "SN2_Step(出口)")
   END_RUNG
   RUNG wire#w1
      Contact( "AutoStep_P" )
   END_RUNG wire#w2
   // the same network as SCL:
   #_w1 := "Auto" AND ("SN2_Step(出口)" = 510);
   #EX_阻挡下降指令[1] := #_w1 AND NOT "EX_阻挡下到位";
   IF #_w1 AND (NOT "AutoStep" OR "AutoStep_P") AND "EX_阻挡下到位" THEN "SN2_Step(出口)" := 515; END_IF;
END_REGION

REGION Network 7: @搬入 电机反转搬入
   RUNG wire#powerrail
      Contact( "Auto" )
      { S7_Templates := "SrcType := Int" } EQ_Contact(in1 := "SN2_Step(出口)", in2 := 515)
      wire#w1
      Coil( "变频器1反转指令自动" )
   END_RUNG
   RUNG wire#w1
      I_Contact( "AutoStep" )
      wire#w2
      Contact( "Com_DB".K03.EX_托盘在席 )
      Move(in := 520, out1 => "SN2_Step(出口)")
   END_RUNG
   RUNG wire#w1
      Contact( "AutoStep_P" )
   END_RUNG wire#w2
   // the same network as SCL:
   "变频器1反转指令自动" := "Auto" AND ("SN2_Step(出口)" = 515);
   IF "变频器1反转指令自动" AND (NOT "AutoStep" OR "AutoStep_P") AND "Com_DB".K03.EX_托盘在席 THEN
       "SN2_Step(出口)" := 520;
   END_IF;
END_REGION

REGION Network 8: @搬入 阻挡上升
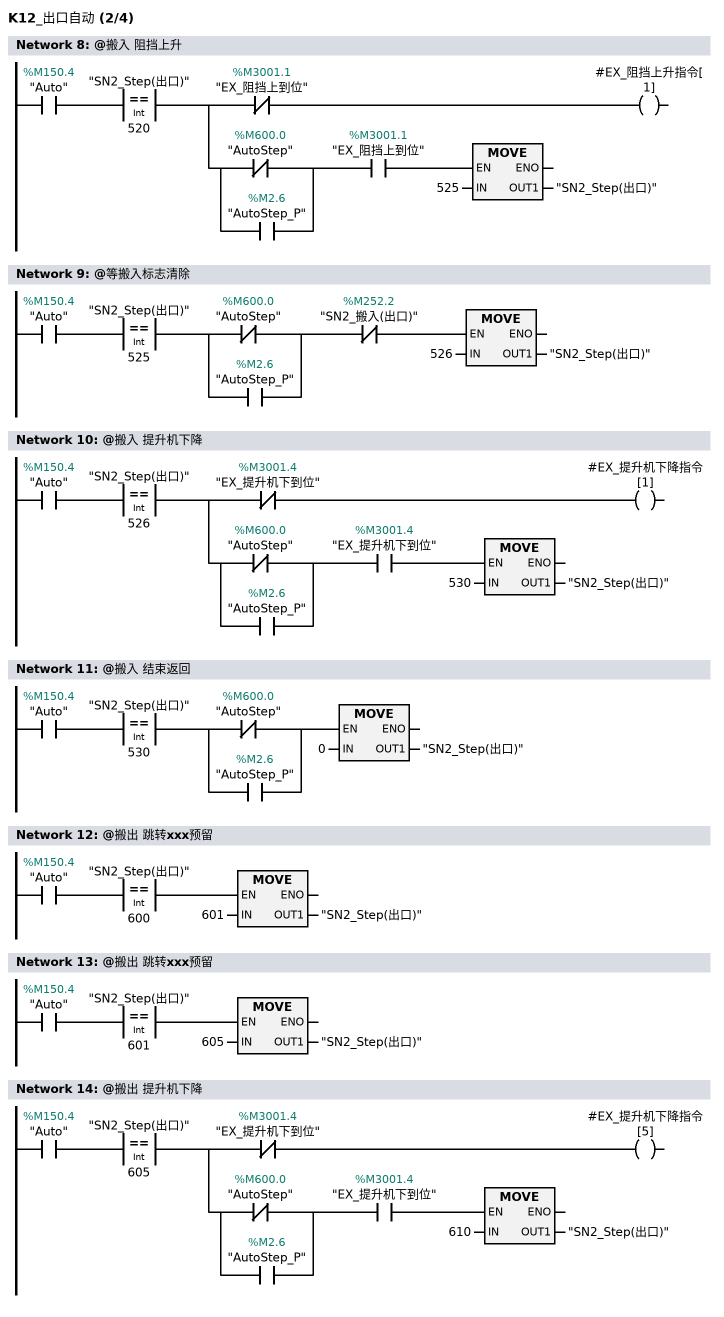
   RUNG wire#powerrail
      Contact( "Auto" )
      { S7_Templates := "SrcType := Int" } EQ_Contact(in1 := "SN2_Step(出口)", in2 := 520)
      wire#w1
      I_Contact( "EX_阻挡上到位" )
      Coil( #EX_阻挡上升指令[1] )
   END_RUNG
   RUNG wire#w1
      I_Contact( "AutoStep" )
      wire#w2
      Contact( "EX_阻挡上到位" )
      Move(in := 525, out1 => "SN2_Step(出口)")
   END_RUNG
   RUNG wire#w1
      Contact( "AutoStep_P" )
   END_RUNG wire#w2
   // the same network as SCL:
   #_w1 := "Auto" AND ("SN2_Step(出口)" = 520);
   #EX_阻挡上升指令[1] := #_w1 AND NOT "EX_阻挡上到位";
   IF #_w1 AND (NOT "AutoStep" OR "AutoStep_P") AND "EX_阻挡上到位" THEN "SN2_Step(出口)" := 525; END_IF;
END_REGION

REGION Network 9: @等搬入标志清除
   RUNG wire#powerrail
      Contact( "Auto" )
      { S7_Templates := "SrcType := Int" } EQ_Contact(in1 := "SN2_Step(出口)", in2 := 525)
      wire#w1
      I_Contact( "AutoStep" )
      wire#w2
      I_Contact( "SN2_搬入(出口)" )
      Move(in := 526, out1 => "SN2_Step(出口)")
   END_RUNG
   RUNG wire#w1
      Contact( "AutoStep_P" )
   END_RUNG wire#w2
   // the same network as SCL:
   IF "Auto" AND ("SN2_Step(出口)" = 525) AND (NOT "AutoStep" OR "AutoStep_P") AND NOT "SN2_搬入(出口)" THEN
       "SN2_Step(出口)" := 526;
   END_IF;
END_REGION

REGION Network 10: @搬入 提升机下降
   RUNG wire#powerrail
      Contact( "Auto" )
      { S7_Templates := "SrcType := Int" } EQ_Contact(in1 := "SN2_Step(出口)", in2 := 526)
      wire#w1
      I_Contact( "EX_提升机下到位" )
      Coil( #EX_提升机下降指令[1] )
   END_RUNG
   RUNG wire#w1
      I_Contact( "AutoStep" )
      wire#w2
      Contact( "EX_提升机下到位" )
      Move(in := 530, out1 => "SN2_Step(出口)")
   END_RUNG
   RUNG wire#w1
      Contact( "AutoStep_P" )
   END_RUNG wire#w2
   // the same network as SCL:
   #_w1 := "Auto" AND ("SN2_Step(出口)" = 526);
   #EX_提升机下降指令[1] := #_w1 AND NOT "EX_提升机下到位";
   IF #_w1 AND (NOT "AutoStep" OR "AutoStep_P") AND "EX_提升机下到位" THEN "SN2_Step(出口)" := 530; END_IF;
END_REGION

REGION Network 11: @搬入 结束返回
   RUNG wire#powerrail
      Contact( "Auto" )
      { S7_Templates := "SrcType := Int" } EQ_Contact(in1 := "SN2_Step(出口)", in2 := 530)
      wire#w1
      I_Contact( "AutoStep" )
      wire#w2
      Move(in := 0, out1 => "SN2_Step(出口)")
   END_RUNG
   RUNG wire#w1
      Contact( "AutoStep_P" )
   END_RUNG wire#w2
   // the same network as SCL:
   IF "Auto" AND ("SN2_Step(出口)" = 530) AND (NOT "AutoStep" OR "AutoStep_P") THEN
       "SN2_Step(出口)" := 0;
   END_IF;
END_REGION

REGION Network 12: @搬出 跳转xxx预留
   RUNG wire#powerrail
      Contact( "Auto" )
      { S7_Templates := "SrcType := Int" } EQ_Contact(in1 := "SN2_Step(出口)", in2 := 600)
      Move(in := 601, out1 => "SN2_Step(出口)")
   END_RUNG
   // the same network as SCL:
   IF "Auto" AND ("SN2_Step(出口)" = 600) THEN "SN2_Step(出口)" := 601; END_IF;
END_REGION

REGION Network 13: @搬出 跳转xxx预留
   RUNG wire#powerrail
      Contact( "Auto" )
      { S7_Templates := "SrcType := Int" } EQ_Contact(in1 := "SN2_Step(出口)", in2 := 601)
      Move(in := 605, out1 => "SN2_Step(出口)")
   END_RUNG
   // the same network as SCL:
   IF "Auto" AND ("SN2_Step(出口)" = 601) THEN "SN2_Step(出口)" := 605; END_IF;
END_REGION

REGION Network 14: @搬出 提升机下降
   RUNG wire#powerrail
      Contact( "Auto" )
      { S7_Templates := "SrcType := Int" } EQ_Contact(in1 := "SN2_Step(出口)", in2 := 605)
      wire#w1
      I_Contact( "EX_提升机下到位" )
      Coil( #EX_提升机下降指令[5] )
   END_RUNG
   RUNG wire#w1
      I_Contact( "AutoStep" )
      wire#w2
      Contact( "EX_提升机下到位" )
      Move(in := 610, out1 => "SN2_Step(出口)")
   END_RUNG
   RUNG wire#w1
      Contact( "AutoStep_P" )
   END_RUNG wire#w2
   // the same network as SCL:
   #_w1 := "Auto" AND ("SN2_Step(出口)" = 605);
   #EX_提升机下降指令[5] := #_w1 AND NOT "EX_提升机下到位";
   IF #_w1 AND (NOT "AutoStep" OR "AutoStep_P") AND "EX_提升机下到位" THEN "SN2_Step(出口)" := 610; END_IF;
END_REGION

REGION Network 15: @搬出 阻挡下降
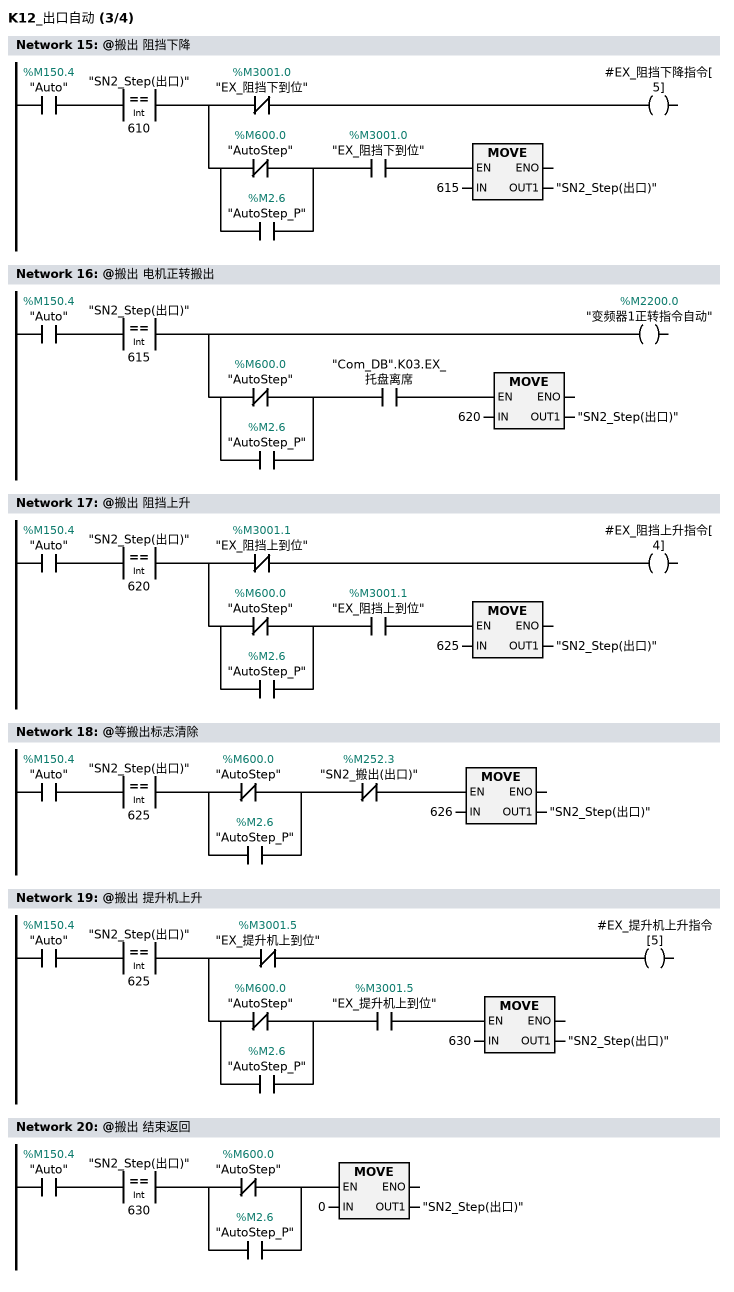
   RUNG wire#powerrail
      Contact( "Auto" )
      { S7_Templates := "SrcType := Int" } EQ_Contact(in1 := "SN2_Step(出口)", in2 := 610)
      wire#w1
      I_Contact( "EX_阻挡下到位" )
      Coil( #EX_阻挡下降指令[5] )
   END_RUNG
   RUNG wire#w1
      I_Contact( "AutoStep" )
      wire#w2
      Contact( "EX_阻挡下到位" )
      Move(in := 615, out1 => "SN2_Step(出口)")
   END_RUNG
   RUNG wire#w1
      Contact( "AutoStep_P" )
   END_RUNG wire#w2
   // the same network as SCL:
   #_w1 := "Auto" AND ("SN2_Step(出口)" = 610);
   #EX_阻挡下降指令[5] := #_w1 AND NOT "EX_阻挡下到位";
   IF #_w1 AND (NOT "AutoStep" OR "AutoStep_P") AND "EX_阻挡下到位" THEN "SN2_Step(出口)" := 615; END_IF;
END_REGION

REGION Network 16: @搬出 电机正转搬出
   RUNG wire#powerrail
      Contact( "Auto" )
      { S7_Templates := "SrcType := Int" } EQ_Contact(in1 := "SN2_Step(出口)", in2 := 615)
      wire#w1
      Coil( "变频器1正转指令自动" )
   END_RUNG
   RUNG wire#w1
      I_Contact( "AutoStep" )
      wire#w2
      Contact( "Com_DB".K03.EX_托盘离席 )
      Move(in := 620, out1 => "SN2_Step(出口)")
   END_RUNG
   RUNG wire#w1
      Contact( "AutoStep_P" )
   END_RUNG wire#w2
   // the same network as SCL:
   "变频器1正转指令自动" := "Auto" AND ("SN2_Step(出口)" = 615);
   IF "变频器1正转指令自动" AND (NOT "AutoStep" OR "AutoStep_P") AND "Com_DB".K03.EX_托盘离席 THEN
       "SN2_Step(出口)" := 620;
   END_IF;
END_REGION

REGION Network 17: @搬出 阻挡上升
   RUNG wire#powerrail
      Contact( "Auto" )
      { S7_Templates := "SrcType := Int" } EQ_Contact(in1 := "SN2_Step(出口)", in2 := 620)
      wire#w1
      I_Contact( "EX_阻挡上到位" )
      Coil( #EX_阻挡上升指令[4] )
   END_RUNG
   RUNG wire#w1
      I_Contact( "AutoStep" )
      wire#w2
      Contact( "EX_阻挡上到位" )
      Move(in := 625, out1 => "SN2_Step(出口)")
   END_RUNG
   RUNG wire#w1
      Contact( "AutoStep_P" )
   END_RUNG wire#w2
   // the same network as SCL:
   #_w1 := "Auto" AND ("SN2_Step(出口)" = 620);
   #EX_阻挡上升指令[4] := #_w1 AND NOT "EX_阻挡上到位";
   IF #_w1 AND (NOT "AutoStep" OR "AutoStep_P") AND "EX_阻挡上到位" THEN "SN2_Step(出口)" := 625; END_IF;
END_REGION

REGION Network 18: @等搬出标志清除
   RUNG wire#powerrail
      Contact( "Auto" )
      { S7_Templates := "SrcType := Int" } EQ_Contact(in1 := "SN2_Step(出口)", in2 := 625)
      wire#w1
      I_Contact( "AutoStep" )
      wire#w2
      I_Contact( "SN2_搬出(出口)" )
      Move(in := 626, out1 => "SN2_Step(出口)")
   END_RUNG
   RUNG wire#w1
      Contact( "AutoStep_P" )
   END_RUNG wire#w2
   // the same network as SCL:
   IF "Auto" AND ("SN2_Step(出口)" = 625) AND (NOT "AutoStep" OR "AutoStep_P") AND NOT "SN2_搬出(出口)" THEN
       "SN2_Step(出口)" := 626;
   END_IF;
END_REGION

REGION Network 19: @搬出 提升机上升
   RUNG wire#powerrail
      Contact( "Auto" )
      { S7_Templates := "SrcType := Int" } EQ_Contact(in1 := "SN2_Step(出口)", in2 := 625)
      wire#w1
      I_Contact( "EX_提升机上到位" )
      Coil( #EX_提升机上升指令[5] )
   END_RUNG
   RUNG wire#w1
      I_Contact( "AutoStep" )
      wire#w2
      Contact( "EX_提升机上到位" )
      Move(in := 630, out1 => "SN2_Step(出口)")
   END_RUNG
   RUNG wire#w1
      Contact( "AutoStep_P" )
   END_RUNG wire#w2
   // the same network as SCL:
   #_w1 := "Auto" AND ("SN2_Step(出口)" = 625);
   #EX_提升机上升指令[5] := #_w1 AND NOT "EX_提升机上到位";
   IF #_w1 AND (NOT "AutoStep" OR "AutoStep_P") AND "EX_提升机上到位" THEN "SN2_Step(出口)" := 630; END_IF;
END_REGION

REGION Network 20: @搬出 结束返回
   RUNG wire#powerrail
      Contact( "Auto" )
      { S7_Templates := "SrcType := Int" } EQ_Contact(in1 := "SN2_Step(出口)", in2 := 630)
      wire#w1
      I_Contact( "AutoStep" )
      wire#w2
      Move(in := 0, out1 => "SN2_Step(出口)")
   END_RUNG
   RUNG wire#w1
      Contact( "AutoStep_P" )
   END_RUNG wire#w2
   // the same network as SCL:
   IF "Auto" AND ("SN2_Step(出口)" = 630) AND (NOT "AutoStep" OR "AutoStep_P") THEN
       "SN2_Step(出口)" := 0;
   END_IF;
END_REGION

REGION Network 21: @控制输出
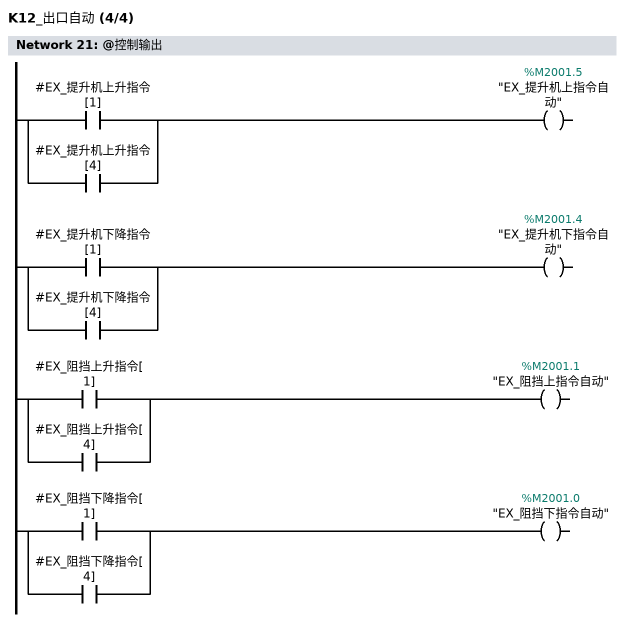
   RUNG wire#powerrail
      Contact( #EX_提升机上升指令[1] )
      wire#w1
      Coil( "EX_提升机上指令自动" )
   END_RUNG
   RUNG wire#powerrail
      Contact( #EX_提升机上升指令[4] )
   END_RUNG wire#w1
   RUNG wire#powerrail
      Contact( #EX_提升机下降指令[1] )
      wire#w2
      Coil( "EX_提升机下指令自动" )
   END_RUNG
   RUNG wire#powerrail
      Contact( #EX_提升机下降指令[4] )
   END_RUNG wire#w2
   RUNG wire#powerrail
      Contact( #EX_阻挡上升指令[1] )
      wire#w3
      Coil( "EX_阻挡上指令自动" )
   END_RUNG
   RUNG wire#powerrail
      Contact( #EX_阻挡上升指令[4] )
   END_RUNG wire#w3
   RUNG wire#powerrail
      Contact( #EX_阻挡下降指令[1] )
      wire#w4
      Coil( "EX_阻挡下指令自动" )
   END_RUNG
   RUNG wire#powerrail
      Contact( #EX_阻挡下降指令[4] )
   END_RUNG wire#w4
   // the same network as SCL:
   "EX_提升机上指令自动" := #EX_提升机上升指令[1] OR #EX_提升机上升指令[4];
   "EX_提升机下指令自动" := #EX_提升机下降指令[1] OR #EX_提升机下降指令[4];
   "EX_阻挡上指令自动" := #EX_阻挡上升指令[1] OR #EX_阻挡上升指令[4];
   "EX_阻挡下指令自动" := #EX_阻挡下降指令[1] OR #EX_阻挡下降指令[4];
END_REGION
END_FUNCTION_BLOCK

FUNCTION_BLOCK "K13_ST01上自动"   // FB13, LAD
{ S7_Optimized_Access := 'TRUE' }
VERSION : 0.1
// stored: AutoNumber false, IsIECCheckEnabled false, IsRetainMemResEnabled false, MemoryReserve 100, SetENOAutomatically false, UDAEnableTagReadback false
   VAR_TEMP   // added for the SCL form of the ladder/FBD networks
      _w1 : Bool;
   END_VAR
BEGIN

REGION Network 1: @搬出条件，SN3===ST01上工位
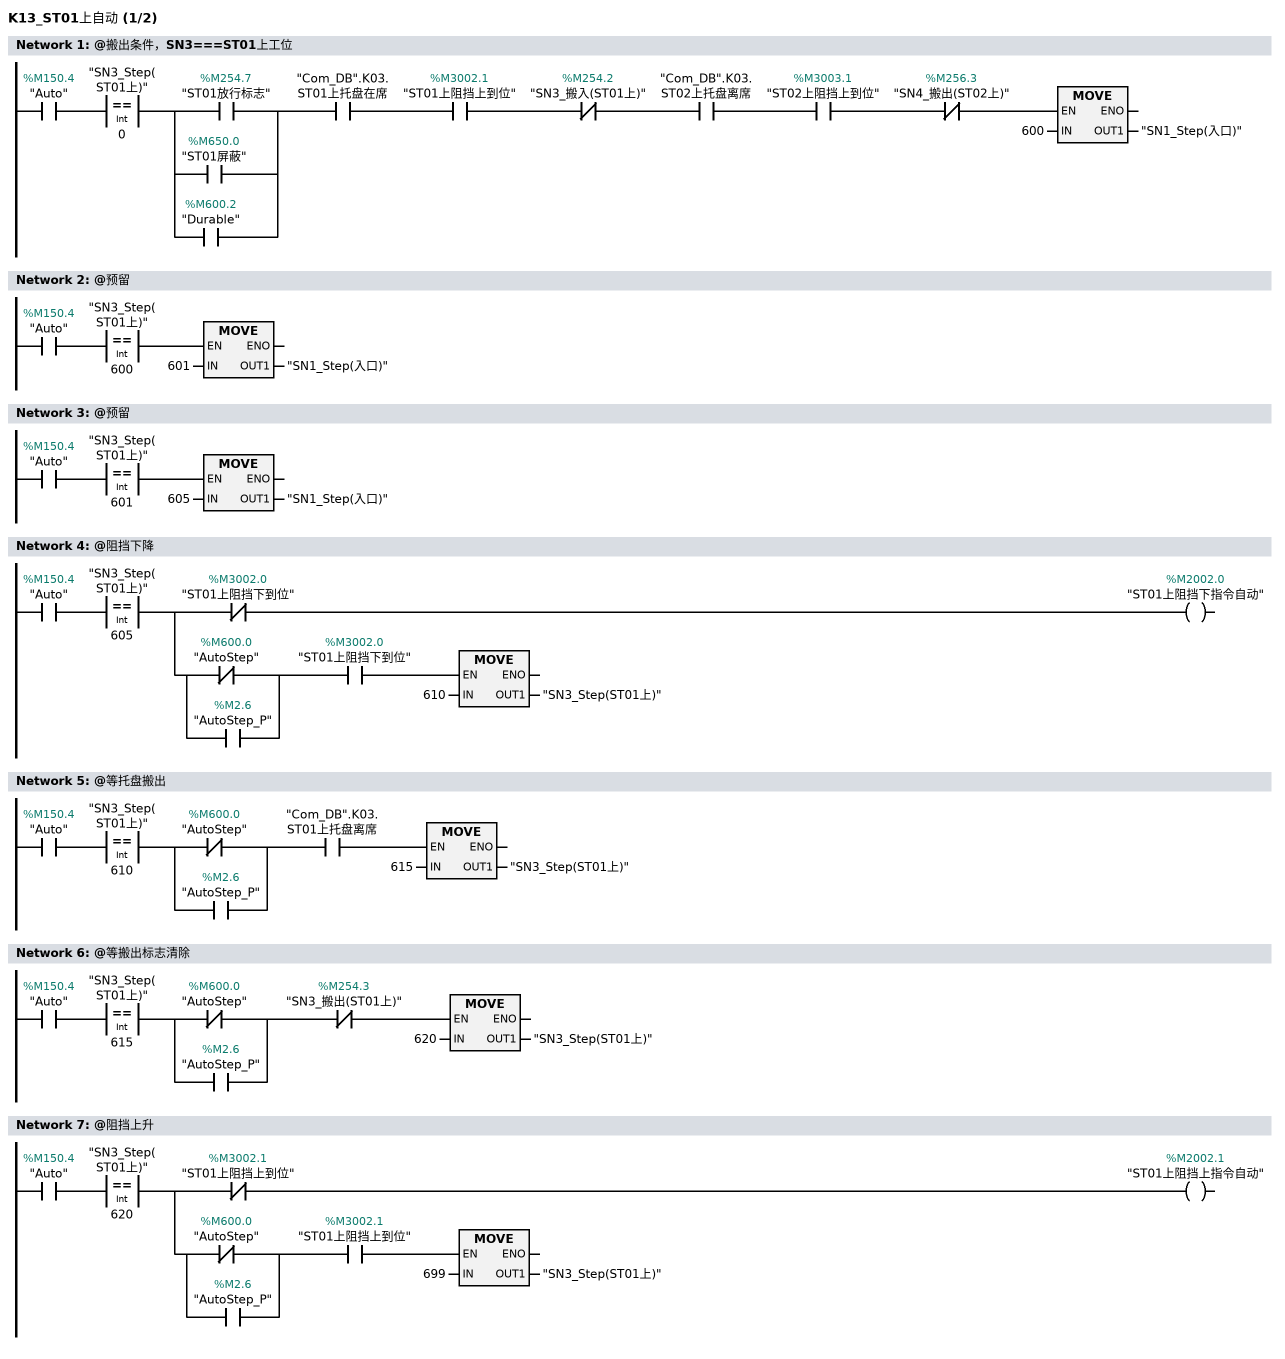
   RUNG wire#powerrail
      Contact( "Auto" )
      { S7_Templates := "SrcType := Int" } EQ_Contact(in1 := "SN3_Step(ST01上)", in2 := 0)
      wire#w1
      Contact( "ST01放行标志" )
      wire#w2
      Contact( "Com_DB".K03.ST01上托盘在席 )
      Contact( "ST01上阻挡上到位" )
      I_Contact( "SN3_搬入(ST01上)" )
      Contact( "Com_DB".K03.ST02上托盘离席 )
      Contact( "ST02上阻挡上到位" )
      I_Contact( "SN4_搬出(ST02上)" )
      Move(in := 600, out1 => "SN1_Step(入口)")
   END_RUNG
   RUNG wire#w1
      Contact( "ST01屏蔽" )
   END_RUNG wire#w2
   RUNG wire#w1
      Contact( "Durable" )
   END_RUNG wire#w2
   // the same network as SCL:
   IF "Auto" AND ("SN3_Step(ST01上)" = 0) AND ("ST01放行标志" OR "ST01屏蔽" OR "Durable") AND "Com_DB".K03.ST01上托盘在席 AND "ST01上阻挡上到位" AND NOT "SN3_搬入(ST01上)" AND "Com_DB".K03.ST02上托盘离席 AND "ST02上阻挡上到位" AND NOT "SN4_搬出(ST02上)" THEN
       "SN1_Step(入口)" := 600;
   END_IF;
END_REGION

REGION Network 2: @预留
   RUNG wire#powerrail
      Contact( "Auto" )
      { S7_Templates := "SrcType := Int" } EQ_Contact(in1 := "SN3_Step(ST01上)", in2 := 600)
      Move(in := 601, out1 => "SN1_Step(入口)")
   END_RUNG
   // the same network as SCL:
   IF "Auto" AND ("SN3_Step(ST01上)" = 600) THEN "SN1_Step(入口)" := 601; END_IF;
END_REGION

REGION Network 3: @预留
   RUNG wire#powerrail
      Contact( "Auto" )
      { S7_Templates := "SrcType := Int" } EQ_Contact(in1 := "SN3_Step(ST01上)", in2 := 601)
      Move(in := 605, out1 => "SN1_Step(入口)")
   END_RUNG
   // the same network as SCL:
   IF "Auto" AND ("SN3_Step(ST01上)" = 601) THEN "SN1_Step(入口)" := 605; END_IF;
END_REGION

REGION Network 4: @阻挡下降
   RUNG wire#powerrail
      Contact( "Auto" )
      { S7_Templates := "SrcType := Int" } EQ_Contact(in1 := "SN3_Step(ST01上)", in2 := 605)
      wire#w1
      I_Contact( "ST01上阻挡下到位" )
      Coil( "ST01上阻挡下指令自动" )
   END_RUNG
   RUNG wire#w1
      I_Contact( "AutoStep" )
      wire#w2
      Contact( "ST01上阻挡下到位" )
      Move(in := 610, out1 => "SN3_Step(ST01上)")
   END_RUNG
   RUNG wire#w1
      Contact( "AutoStep_P" )
   END_RUNG wire#w2
   // the same network as SCL:
   #_w1 := "Auto" AND ("SN3_Step(ST01上)" = 605);
   "ST01上阻挡下指令自动" := #_w1 AND NOT "ST01上阻挡下到位";
   IF #_w1 AND (NOT "AutoStep" OR "AutoStep_P") AND "ST01上阻挡下到位" THEN "SN3_Step(ST01上)" := 610; END_IF;
END_REGION

REGION Network 5: @等托盘搬出
   RUNG wire#powerrail
      Contact( "Auto" )
      { S7_Templates := "SrcType := Int" } EQ_Contact(in1 := "SN3_Step(ST01上)", in2 := 610)
      wire#w1
      I_Contact( "AutoStep" )
      wire#w2
      Contact( "Com_DB".K03.ST01上托盘离席 )
      Move(in := 615, out1 => "SN3_Step(ST01上)")
   END_RUNG
   RUNG wire#w1
      Contact( "AutoStep_P" )
   END_RUNG wire#w2
   // the same network as SCL:
   IF "Auto" AND ("SN3_Step(ST01上)" = 610) AND (NOT "AutoStep" OR "AutoStep_P") AND "Com_DB".K03.ST01上托盘离席 THEN
       "SN3_Step(ST01上)" := 615;
   END_IF;
END_REGION

REGION Network 6: @等搬出标志清除
   RUNG wire#powerrail
      Contact( "Auto" )
      { S7_Templates := "SrcType := Int" } EQ_Contact(in1 := "SN3_Step(ST01上)", in2 := 615)
      wire#w1
      I_Contact( "AutoStep" )
      wire#w2
      I_Contact( "SN3_搬出(ST01上)" )
      Move(in := 620, out1 => "SN3_Step(ST01上)")
   END_RUNG
   RUNG wire#w1
      Contact( "AutoStep_P" )
   END_RUNG wire#w2
   // the same network as SCL:
   IF "Auto" AND ("SN3_Step(ST01上)" = 615) AND (NOT "AutoStep" OR "AutoStep_P") AND NOT "SN3_搬出(ST01上)" THEN
       "SN3_Step(ST01上)" := 620;
   END_IF;
END_REGION

REGION Network 7: @阻挡上升
   RUNG wire#powerrail
      Contact( "Auto" )
      { S7_Templates := "SrcType := Int" } EQ_Contact(in1 := "SN3_Step(ST01上)", in2 := 620)
      wire#w1
      I_Contact( "ST01上阻挡上到位" )
      Coil( "ST01上阻挡上指令自动" )
   END_RUNG
   RUNG wire#w1
      I_Contact( "AutoStep" )
      wire#w2
      Contact( "ST01上阻挡上到位" )
      Move(in := 699, out1 => "SN3_Step(ST01上)")
   END_RUNG
   RUNG wire#w1
      Contact( "AutoStep_P" )
   END_RUNG wire#w2
   // the same network as SCL:
   #_w1 := "Auto" AND ("SN3_Step(ST01上)" = 620);
   "ST01上阻挡上指令自动" := #_w1 AND NOT "ST01上阻挡上到位";
   IF #_w1 AND (NOT "AutoStep" OR "AutoStep_P") AND "ST01上阻挡上到位" THEN "SN3_Step(ST01上)" := 699; END_IF;
END_REGION

REGION Network 8: @返回
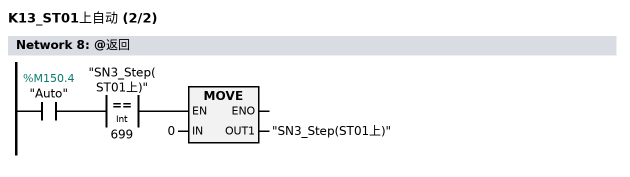
   RUNG wire#powerrail
      Contact( "Auto" )
      { S7_Templates := "SrcType := Int" } EQ_Contact(in1 := "SN3_Step(ST01上)", in2 := 699)
      Move(in := 0, out1 => "SN3_Step(ST01上)")
   END_RUNG
   // the same network as SCL:
   IF "Auto" AND ("SN3_Step(ST01上)" = 699) THEN "SN3_Step(ST01上)" := 0; END_IF;
END_REGION
END_FUNCTION_BLOCK

FUNCTION_BLOCK "K14_ST02上自动"   // FB14, LAD
{ S7_Optimized_Access := 'TRUE' }
VERSION : 0.1
// stored: AutoNumber false, IsIECCheckEnabled false, IsRetainMemResEnabled false, MemoryReserve 100, SetENOAutomatically false, UDAEnableTagReadback false
   VAR_TEMP   // added for the SCL form of the ladder/FBD networks
      _w1 : Bool;
   END_VAR
BEGIN

REGION Network 2: @搬出条件，SN4===ST02上工位
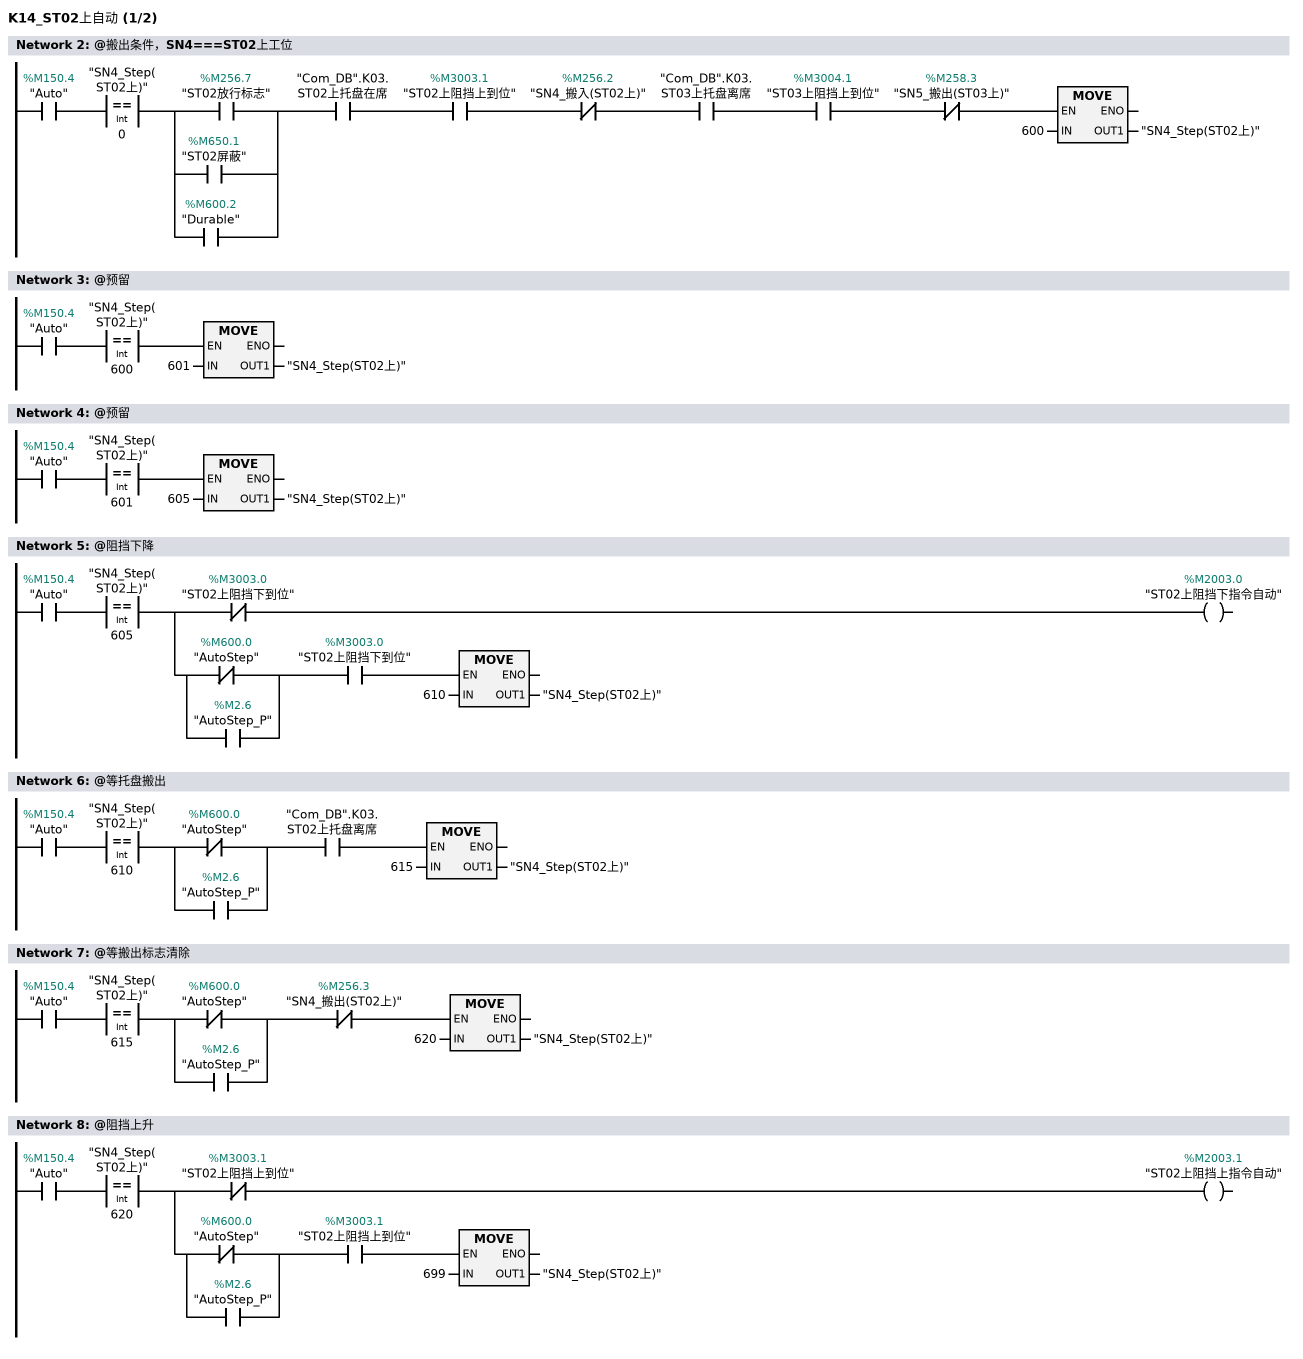
   RUNG wire#powerrail
      Contact( "Auto" )
      { S7_Templates := "SrcType := Int" } EQ_Contact(in1 := "SN4_Step(ST02上)", in2 := 0)
      wire#w1
      Contact( "ST02放行标志" )
      wire#w2
      Contact( "Com_DB".K03.ST02上托盘在席 )
      Contact( "ST02上阻挡上到位" )
      I_Contact( "SN4_搬入(ST02上)" )
      Contact( "Com_DB".K03.ST03上托盘离席 )
      Contact( "ST03上阻挡上到位" )
      I_Contact( "SN5_搬出(ST03上)" )
      Move(in := 600, out1 => "SN4_Step(ST02上)")
   END_RUNG
   RUNG wire#w1
      Contact( "ST02屏蔽" )
   END_RUNG wire#w2
   RUNG wire#w1
      Contact( "Durable" )
   END_RUNG wire#w2
   // the same network as SCL:
   IF "Auto" AND ("SN4_Step(ST02上)" = 0) AND ("ST02放行标志" OR "ST02屏蔽" OR "Durable") AND "Com_DB".K03.ST02上托盘在席 AND "ST02上阻挡上到位" AND NOT "SN4_搬入(ST02上)" AND "Com_DB".K03.ST03上托盘离席 AND "ST03上阻挡上到位" AND NOT "SN5_搬出(ST03上)" THEN
       "SN4_Step(ST02上)" := 600;
   END_IF;
END_REGION

REGION Network 3: @预留
   RUNG wire#powerrail
      Contact( "Auto" )
      { S7_Templates := "SrcType := Int" } EQ_Contact(in1 := "SN4_Step(ST02上)", in2 := 600)
      Move(in := 601, out1 => "SN4_Step(ST02上)")
   END_RUNG
   // the same network as SCL:
   IF "Auto" AND ("SN4_Step(ST02上)" = 600) THEN "SN4_Step(ST02上)" := 601; END_IF;
END_REGION

REGION Network 4: @预留
   RUNG wire#powerrail
      Contact( "Auto" )
      { S7_Templates := "SrcType := Int" } EQ_Contact(in1 := "SN4_Step(ST02上)", in2 := 601)
      Move(in := 605, out1 => "SN4_Step(ST02上)")
   END_RUNG
   // the same network as SCL:
   IF "Auto" AND ("SN4_Step(ST02上)" = 601) THEN "SN4_Step(ST02上)" := 605; END_IF;
END_REGION

REGION Network 5: @阻挡下降
   RUNG wire#powerrail
      Contact( "Auto" )
      { S7_Templates := "SrcType := Int" } EQ_Contact(in1 := "SN4_Step(ST02上)", in2 := 605)
      wire#w1
      I_Contact( "ST02上阻挡下到位" )
      Coil( "ST02上阻挡下指令自动" )
   END_RUNG
   RUNG wire#w1
      I_Contact( "AutoStep" )
      wire#w2
      Contact( "ST02上阻挡下到位" )
      Move(in := 610, out1 => "SN4_Step(ST02上)")
   END_RUNG
   RUNG wire#w1
      Contact( "AutoStep_P" )
   END_RUNG wire#w2
   // the same network as SCL:
   #_w1 := "Auto" AND ("SN4_Step(ST02上)" = 605);
   "ST02上阻挡下指令自动" := #_w1 AND NOT "ST02上阻挡下到位";
   IF #_w1 AND (NOT "AutoStep" OR "AutoStep_P") AND "ST02上阻挡下到位" THEN "SN4_Step(ST02上)" := 610; END_IF;
END_REGION

REGION Network 6: @等托盘搬出
   RUNG wire#powerrail
      Contact( "Auto" )
      { S7_Templates := "SrcType := Int" } EQ_Contact(in1 := "SN4_Step(ST02上)", in2 := 610)
      wire#w1
      I_Contact( "AutoStep" )
      wire#w2
      Contact( "Com_DB".K03.ST02上托盘离席 )
      Move(in := 615, out1 => "SN4_Step(ST02上)")
   END_RUNG
   RUNG wire#w1
      Contact( "AutoStep_P" )
   END_RUNG wire#w2
   // the same network as SCL:
   IF "Auto" AND ("SN4_Step(ST02上)" = 610) AND (NOT "AutoStep" OR "AutoStep_P") AND "Com_DB".K03.ST02上托盘离席 THEN
       "SN4_Step(ST02上)" := 615;
   END_IF;
END_REGION

REGION Network 7: @等搬出标志清除
   RUNG wire#powerrail
      Contact( "Auto" )
      { S7_Templates := "SrcType := Int" } EQ_Contact(in1 := "SN4_Step(ST02上)", in2 := 615)
      wire#w1
      I_Contact( "AutoStep" )
      wire#w2
      I_Contact( "SN4_搬出(ST02上)" )
      Move(in := 620, out1 => "SN4_Step(ST02上)")
   END_RUNG
   RUNG wire#w1
      Contact( "AutoStep_P" )
   END_RUNG wire#w2
   // the same network as SCL:
   IF "Auto" AND ("SN4_Step(ST02上)" = 615) AND (NOT "AutoStep" OR "AutoStep_P") AND NOT "SN4_搬出(ST02上)" THEN
       "SN4_Step(ST02上)" := 620;
   END_IF;
END_REGION

REGION Network 8: @阻挡上升
   RUNG wire#powerrail
      Contact( "Auto" )
      { S7_Templates := "SrcType := Int" } EQ_Contact(in1 := "SN4_Step(ST02上)", in2 := 620)
      wire#w1
      I_Contact( "ST02上阻挡上到位" )
      Coil( "ST02上阻挡上指令自动" )
   END_RUNG
   RUNG wire#w1
      I_Contact( "AutoStep" )
      wire#w2
      Contact( "ST02上阻挡上到位" )
      Move(in := 699, out1 => "SN4_Step(ST02上)")
   END_RUNG
   RUNG wire#w1
      Contact( "AutoStep_P" )
   END_RUNG wire#w2
   // the same network as SCL:
   #_w1 := "Auto" AND ("SN4_Step(ST02上)" = 620);
   "ST02上阻挡上指令自动" := #_w1 AND NOT "ST02上阻挡上到位";
   IF #_w1 AND (NOT "AutoStep" OR "AutoStep_P") AND "ST02上阻挡上到位" THEN "SN4_Step(ST02上)" := 699; END_IF;
END_REGION

REGION Network 9: @返回
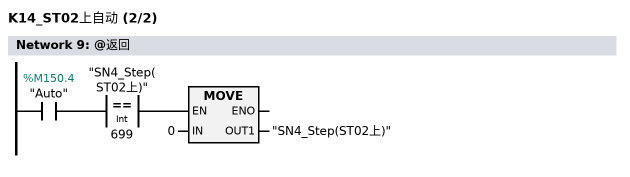
   RUNG wire#powerrail
      Contact( "Auto" )
      { S7_Templates := "SrcType := Int" } EQ_Contact(in1 := "SN4_Step(ST02上)", in2 := 699)
      Move(in := 0, out1 => "SN4_Step(ST02上)")
   END_RUNG
   // the same network as SCL:
   IF "Auto" AND ("SN4_Step(ST02上)" = 699) THEN "SN4_Step(ST02上)" := 0; END_IF;
END_REGION
END_FUNCTION_BLOCK

FUNCTION_BLOCK "K15_ST03上自动"   // FB15, LAD
{ S7_Optimized_Access := 'TRUE' }
VERSION : 0.1
// stored: AutoNumber false, IsIECCheckEnabled false, IsRetainMemResEnabled false, MemoryReserve 100, SetENOAutomatically false, UDAEnableTagReadback false
   VAR_TEMP   // added for the SCL form of the ladder/FBD networks
      _w1 : Bool;
   END_VAR
BEGIN

REGION Network 2: @搬出条件，SN5===ST03上工位
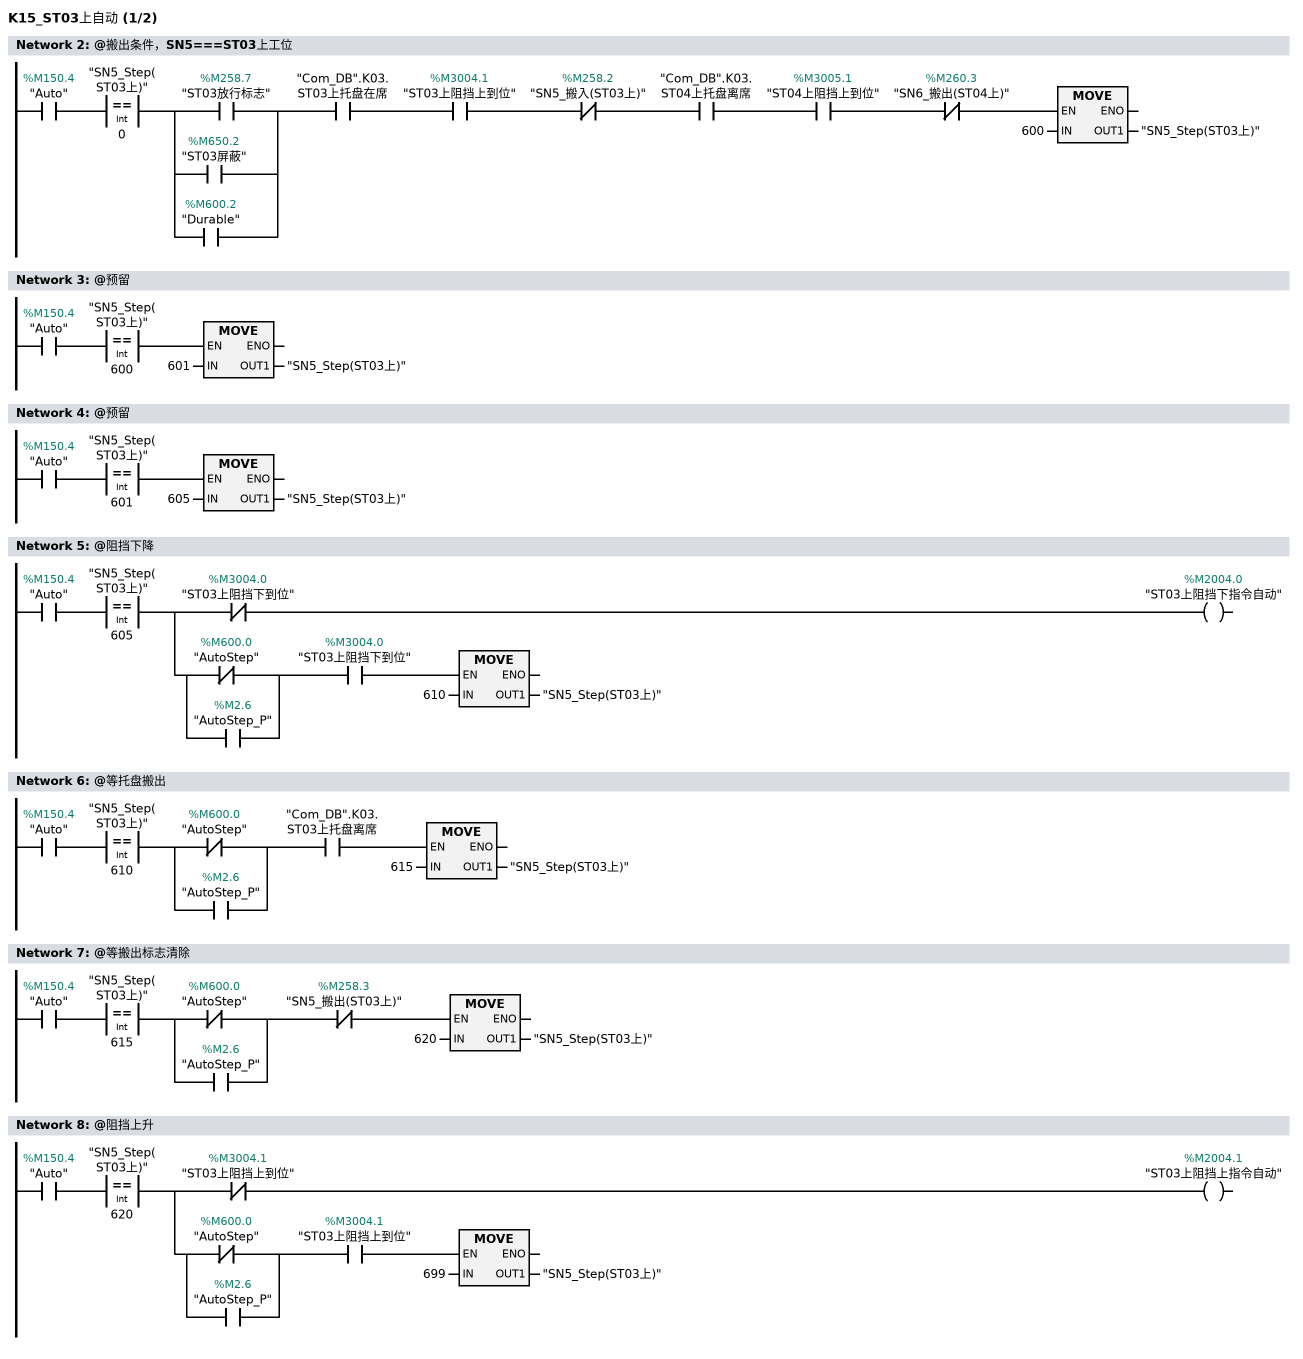
   RUNG wire#powerrail
      Contact( "Auto" )
      { S7_Templates := "SrcType := Int" } EQ_Contact(in1 := "SN5_Step(ST03上)", in2 := 0)
      wire#w1
      Contact( "ST03放行标志" )
      wire#w2
      Contact( "Com_DB".K03.ST03上托盘在席 )
      Contact( "ST03上阻挡上到位" )
      I_Contact( "SN5_搬入(ST03上)" )
      Contact( "Com_DB".K03.ST04上托盘离席 )
      Contact( "ST04上阻挡上到位" )
      I_Contact( "SN6_搬出(ST04上)" )
      Move(in := 600, out1 => "SN5_Step(ST03上)")
   END_RUNG
   RUNG wire#w1
      Contact( "ST03屏蔽" )
   END_RUNG wire#w2
   RUNG wire#w1
      Contact( "Durable" )
   END_RUNG wire#w2
   // the same network as SCL:
   IF "Auto" AND ("SN5_Step(ST03上)" = 0) AND ("ST03放行标志" OR "ST03屏蔽" OR "Durable") AND "Com_DB".K03.ST03上托盘在席 AND "ST03上阻挡上到位" AND NOT "SN5_搬入(ST03上)" AND "Com_DB".K03.ST04上托盘离席 AND "ST04上阻挡上到位" AND NOT "SN6_搬出(ST04上)" THEN
       "SN5_Step(ST03上)" := 600;
   END_IF;
END_REGION

REGION Network 3: @预留
   RUNG wire#powerrail
      Contact( "Auto" )
      { S7_Templates := "SrcType := Int" } EQ_Contact(in1 := "SN5_Step(ST03上)", in2 := 600)
      Move(in := 601, out1 => "SN5_Step(ST03上)")
   END_RUNG
   // the same network as SCL:
   IF "Auto" AND ("SN5_Step(ST03上)" = 600) THEN "SN5_Step(ST03上)" := 601; END_IF;
END_REGION

REGION Network 4: @预留
   RUNG wire#powerrail
      Contact( "Auto" )
      { S7_Templates := "SrcType := Int" } EQ_Contact(in1 := "SN5_Step(ST03上)", in2 := 601)
      Move(in := 605, out1 => "SN5_Step(ST03上)")
   END_RUNG
   // the same network as SCL:
   IF "Auto" AND ("SN5_Step(ST03上)" = 601) THEN "SN5_Step(ST03上)" := 605; END_IF;
END_REGION

REGION Network 5: @阻挡下降
   RUNG wire#powerrail
      Contact( "Auto" )
      { S7_Templates := "SrcType := Int" } EQ_Contact(in1 := "SN5_Step(ST03上)", in2 := 605)
      wire#w1
      I_Contact( "ST03上阻挡下到位" )
      Coil( "ST03上阻挡下指令自动" )
   END_RUNG
   RUNG wire#w1
      I_Contact( "AutoStep" )
      wire#w2
      Contact( "ST03上阻挡下到位" )
      Move(in := 610, out1 => "SN5_Step(ST03上)")
   END_RUNG
   RUNG wire#w1
      Contact( "AutoStep_P" )
   END_RUNG wire#w2
   // the same network as SCL:
   #_w1 := "Auto" AND ("SN5_Step(ST03上)" = 605);
   "ST03上阻挡下指令自动" := #_w1 AND NOT "ST03上阻挡下到位";
   IF #_w1 AND (NOT "AutoStep" OR "AutoStep_P") AND "ST03上阻挡下到位" THEN "SN5_Step(ST03上)" := 610; END_IF;
END_REGION

REGION Network 6: @等托盘搬出
   RUNG wire#powerrail
      Contact( "Auto" )
      { S7_Templates := "SrcType := Int" } EQ_Contact(in1 := "SN5_Step(ST03上)", in2 := 610)
      wire#w1
      I_Contact( "AutoStep" )
      wire#w2
      Contact( "Com_DB".K03.ST03上托盘离席 )
      Move(in := 615, out1 => "SN5_Step(ST03上)")
   END_RUNG
   RUNG wire#w1
      Contact( "AutoStep_P" )
   END_RUNG wire#w2
   // the same network as SCL:
   IF "Auto" AND ("SN5_Step(ST03上)" = 610) AND (NOT "AutoStep" OR "AutoStep_P") AND "Com_DB".K03.ST03上托盘离席 THEN
       "SN5_Step(ST03上)" := 615;
   END_IF;
END_REGION

REGION Network 7: @等搬出标志清除
   RUNG wire#powerrail
      Contact( "Auto" )
      { S7_Templates := "SrcType := Int" } EQ_Contact(in1 := "SN5_Step(ST03上)", in2 := 615)
      wire#w1
      I_Contact( "AutoStep" )
      wire#w2
      I_Contact( "SN5_搬出(ST03上)" )
      Move(in := 620, out1 => "SN5_Step(ST03上)")
   END_RUNG
   RUNG wire#w1
      Contact( "AutoStep_P" )
   END_RUNG wire#w2
   // the same network as SCL:
   IF "Auto" AND ("SN5_Step(ST03上)" = 615) AND (NOT "AutoStep" OR "AutoStep_P") AND NOT "SN5_搬出(ST03上)" THEN
       "SN5_Step(ST03上)" := 620;
   END_IF;
END_REGION

REGION Network 8: @阻挡上升
   RUNG wire#powerrail
      Contact( "Auto" )
      { S7_Templates := "SrcType := Int" } EQ_Contact(in1 := "SN5_Step(ST03上)", in2 := 620)
      wire#w1
      I_Contact( "ST03上阻挡上到位" )
      Coil( "ST03上阻挡上指令自动" )
   END_RUNG
   RUNG wire#w1
      I_Contact( "AutoStep" )
      wire#w2
      Contact( "ST03上阻挡上到位" )
      Move(in := 699, out1 => "SN5_Step(ST03上)")
   END_RUNG
   RUNG wire#w1
      Contact( "AutoStep_P" )
   END_RUNG wire#w2
   // the same network as SCL:
   #_w1 := "Auto" AND ("SN5_Step(ST03上)" = 620);
   "ST03上阻挡上指令自动" := #_w1 AND NOT "ST03上阻挡上到位";
   IF #_w1 AND (NOT "AutoStep" OR "AutoStep_P") AND "ST03上阻挡上到位" THEN "SN5_Step(ST03上)" := 699; END_IF;
END_REGION

REGION Network 9: @返回
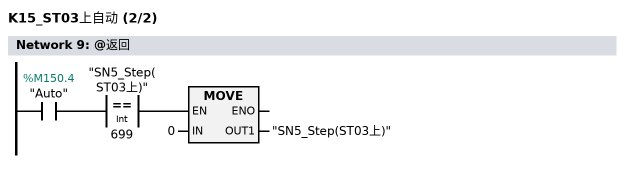
   RUNG wire#powerrail
      Contact( "Auto" )
      { S7_Templates := "SrcType := Int" } EQ_Contact(in1 := "SN5_Step(ST03上)", in2 := 699)
      Move(in := 0, out1 => "SN5_Step(ST03上)")
   END_RUNG
   // the same network as SCL:
   IF "Auto" AND ("SN5_Step(ST03上)" = 699) THEN "SN5_Step(ST03上)" := 0; END_IF;
END_REGION
END_FUNCTION_BLOCK

FUNCTION_BLOCK "K16_ST04上自动"   // FB16, LAD
{ S7_Optimized_Access := 'TRUE' }
VERSION : 0.1
// stored: AutoNumber false, IsIECCheckEnabled false, IsRetainMemResEnabled false, MemoryReserve 100, SetENOAutomatically false, UDAEnableTagReadback false
   VAR_TEMP   // added for the SCL form of the ladder/FBD networks
      _w1 : Bool;
   END_VAR
BEGIN

REGION Network 2: @搬出条件，SN6===ST04上工位
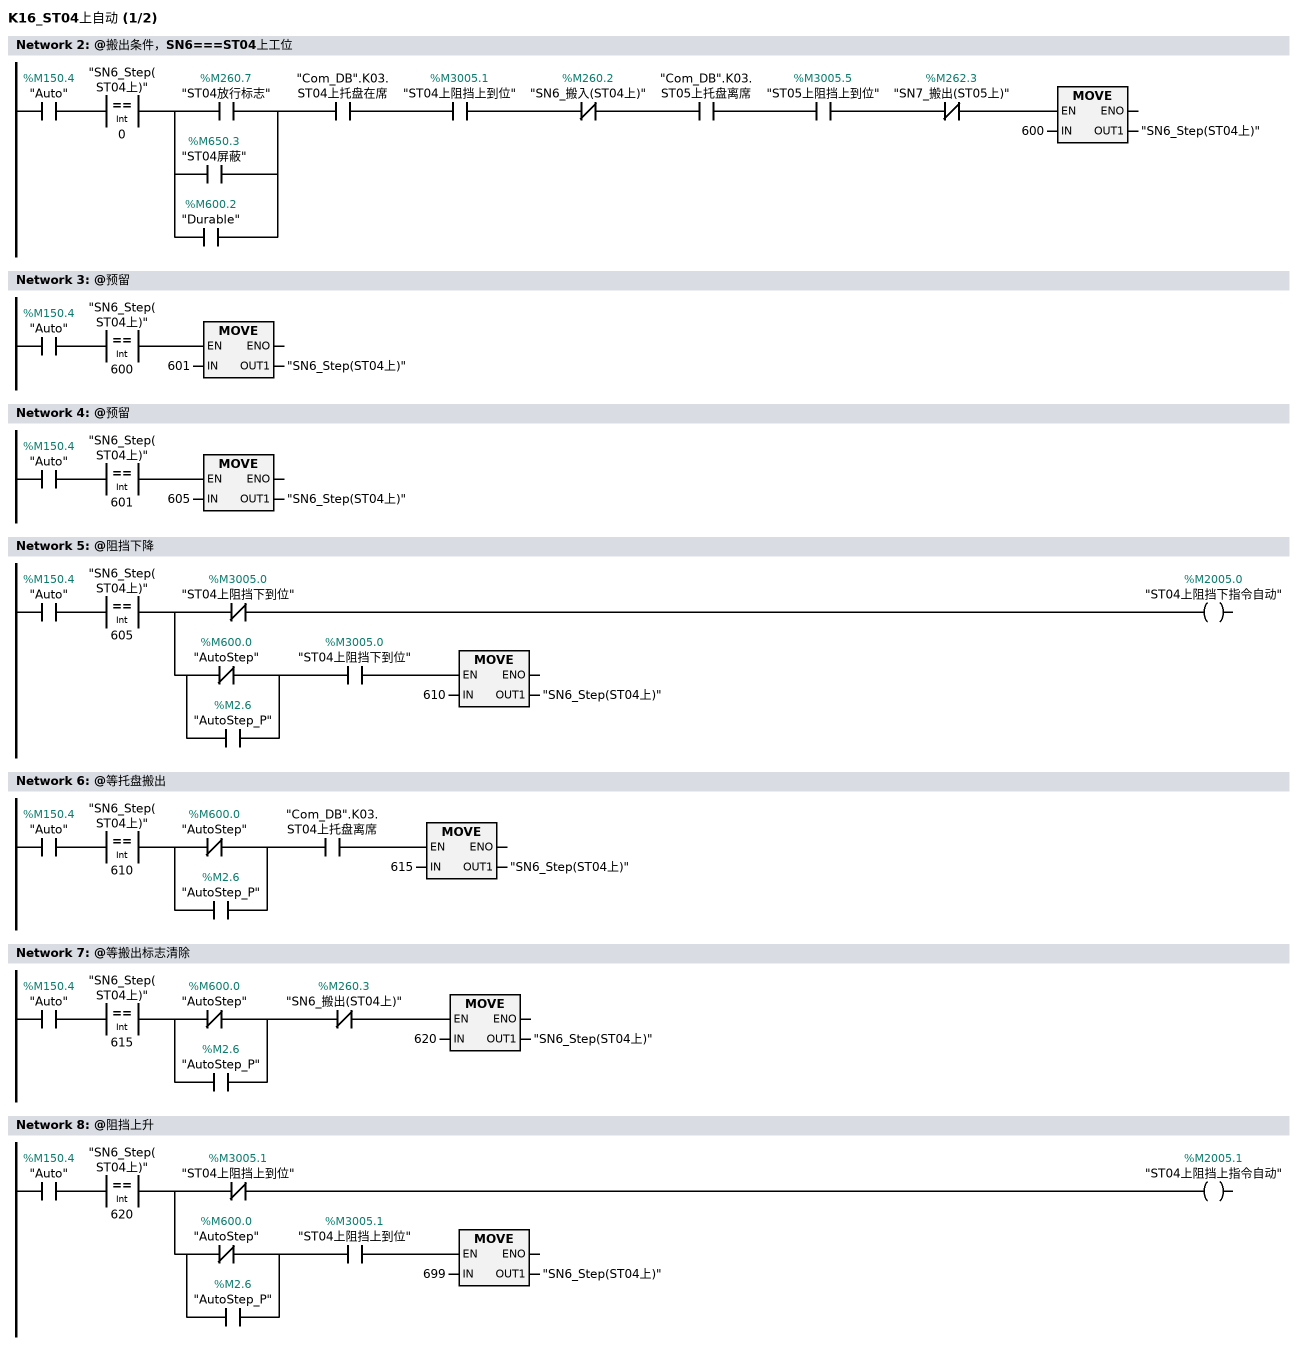
   RUNG wire#powerrail
      Contact( "Auto" )
      { S7_Templates := "SrcType := Int" } EQ_Contact(in1 := "SN6_Step(ST04上)", in2 := 0)
      wire#w1
      Contact( "ST04放行标志" )
      wire#w2
      Contact( "Com_DB".K03.ST04上托盘在席 )
      Contact( "ST04上阻挡上到位" )
      I_Contact( "SN6_搬入(ST04上)" )
      Contact( "Com_DB".K03.ST05上托盘离席 )
      Contact( "ST05上阻挡上到位" )
      I_Contact( "SN7_搬出(ST05上)" )
      Move(in := 600, out1 => "SN6_Step(ST04上)")
   END_RUNG
   RUNG wire#w1
      Contact( "ST04屏蔽" )
   END_RUNG wire#w2
   RUNG wire#w1
      Contact( "Durable" )
   END_RUNG wire#w2
   // the same network as SCL:
   IF "Auto" AND ("SN6_Step(ST04上)" = 0) AND ("ST04放行标志" OR "ST04屏蔽" OR "Durable") AND "Com_DB".K03.ST04上托盘在席 AND "ST04上阻挡上到位" AND NOT "SN6_搬入(ST04上)" AND "Com_DB".K03.ST05上托盘离席 AND "ST05上阻挡上到位" AND NOT "SN7_搬出(ST05上)" THEN
       "SN6_Step(ST04上)" := 600;
   END_IF;
END_REGION

REGION Network 3: @预留
   RUNG wire#powerrail
      Contact( "Auto" )
      { S7_Templates := "SrcType := Int" } EQ_Contact(in1 := "SN6_Step(ST04上)", in2 := 600)
      Move(in := 601, out1 => "SN6_Step(ST04上)")
   END_RUNG
   // the same network as SCL:
   IF "Auto" AND ("SN6_Step(ST04上)" = 600) THEN "SN6_Step(ST04上)" := 601; END_IF;
END_REGION

REGION Network 4: @预留
   RUNG wire#powerrail
      Contact( "Auto" )
      { S7_Templates := "SrcType := Int" } EQ_Contact(in1 := "SN6_Step(ST04上)", in2 := 601)
      Move(in := 605, out1 => "SN6_Step(ST04上)")
   END_RUNG
   // the same network as SCL:
   IF "Auto" AND ("SN6_Step(ST04上)" = 601) THEN "SN6_Step(ST04上)" := 605; END_IF;
END_REGION

REGION Network 5: @阻挡下降
   RUNG wire#powerrail
      Contact( "Auto" )
      { S7_Templates := "SrcType := Int" } EQ_Contact(in1 := "SN6_Step(ST04上)", in2 := 605)
      wire#w1
      I_Contact( "ST04上阻挡下到位" )
      Coil( "ST04上阻挡下指令自动" )
   END_RUNG
   RUNG wire#w1
      I_Contact( "AutoStep" )
      wire#w2
      Contact( "ST04上阻挡下到位" )
      Move(in := 610, out1 => "SN6_Step(ST04上)")
   END_RUNG
   RUNG wire#w1
      Contact( "AutoStep_P" )
   END_RUNG wire#w2
   // the same network as SCL:
   #_w1 := "Auto" AND ("SN6_Step(ST04上)" = 605);
   "ST04上阻挡下指令自动" := #_w1 AND NOT "ST04上阻挡下到位";
   IF #_w1 AND (NOT "AutoStep" OR "AutoStep_P") AND "ST04上阻挡下到位" THEN "SN6_Step(ST04上)" := 610; END_IF;
END_REGION

REGION Network 6: @等托盘搬出
   RUNG wire#powerrail
      Contact( "Auto" )
      { S7_Templates := "SrcType := Int" } EQ_Contact(in1 := "SN6_Step(ST04上)", in2 := 610)
      wire#w1
      I_Contact( "AutoStep" )
      wire#w2
      Contact( "Com_DB".K03.ST04上托盘离席 )
      Move(in := 615, out1 => "SN6_Step(ST04上)")
   END_RUNG
   RUNG wire#w1
      Contact( "AutoStep_P" )
   END_RUNG wire#w2
   // the same network as SCL:
   IF "Auto" AND ("SN6_Step(ST04上)" = 610) AND (NOT "AutoStep" OR "AutoStep_P") AND "Com_DB".K03.ST04上托盘离席 THEN
       "SN6_Step(ST04上)" := 615;
   END_IF;
END_REGION

REGION Network 7: @等搬出标志清除
   RUNG wire#powerrail
      Contact( "Auto" )
      { S7_Templates := "SrcType := Int" } EQ_Contact(in1 := "SN6_Step(ST04上)", in2 := 615)
      wire#w1
      I_Contact( "AutoStep" )
      wire#w2
      I_Contact( "SN6_搬出(ST04上)" )
      Move(in := 620, out1 => "SN6_Step(ST04上)")
   END_RUNG
   RUNG wire#w1
      Contact( "AutoStep_P" )
   END_RUNG wire#w2
   // the same network as SCL:
   IF "Auto" AND ("SN6_Step(ST04上)" = 615) AND (NOT "AutoStep" OR "AutoStep_P") AND NOT "SN6_搬出(ST04上)" THEN
       "SN6_Step(ST04上)" := 620;
   END_IF;
END_REGION

REGION Network 8: @阻挡上升
   RUNG wire#powerrail
      Contact( "Auto" )
      { S7_Templates := "SrcType := Int" } EQ_Contact(in1 := "SN6_Step(ST04上)", in2 := 620)
      wire#w1
      I_Contact( "ST04上阻挡上到位" )
      Coil( "ST04上阻挡上指令自动" )
   END_RUNG
   RUNG wire#w1
      I_Contact( "AutoStep" )
      wire#w2
      Contact( "ST04上阻挡上到位" )
      Move(in := 699, out1 => "SN6_Step(ST04上)")
   END_RUNG
   RUNG wire#w1
      Contact( "AutoStep_P" )
   END_RUNG wire#w2
   // the same network as SCL:
   #_w1 := "Auto" AND ("SN6_Step(ST04上)" = 620);
   "ST04上阻挡上指令自动" := #_w1 AND NOT "ST04上阻挡上到位";
   IF #_w1 AND (NOT "AutoStep" OR "AutoStep_P") AND "ST04上阻挡上到位" THEN "SN6_Step(ST04上)" := 699; END_IF;
END_REGION

REGION Network 9: @返回
